KUKA KRL program: EPS_2_26115_SA6997_A_20260219035528.src

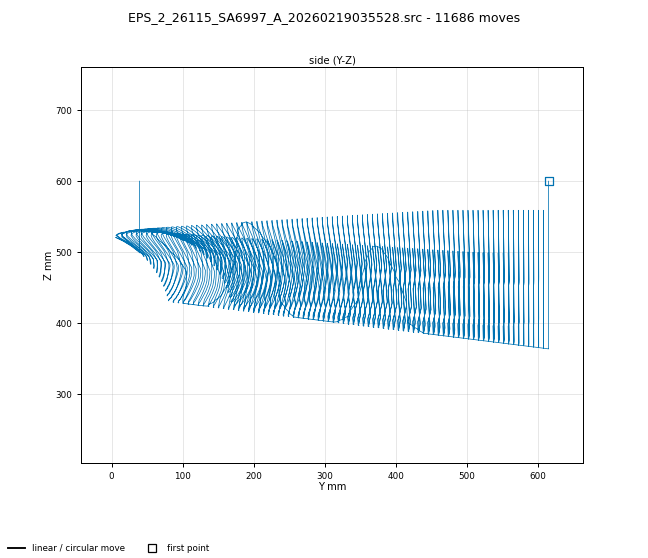
[picture p0: tool path of EPS_2_26115_SA6997_A_20260219035528.src, 11686 of 11688 moves have a stored position in this frame; points joined in program order, loops and branches not executed]
&ACCESS RVP
&REL 4
&COMMENT QRS 19112012
&PARAM EDITMASK = *
DEF PART()
EXT BAS (BAS_COMMAND :IN,REAL :IN )
INT I
BAS (#INITMOV,0 )

;KUKA QRS Post kuka4.cps  Date:22-06-2017 !

File_ID=3052

QRS_PRE_INIT()

;Init var - Until changes are made in qrs_pre_init
Outlet_Square_prg=0
Inlet_1_Square_prg=0
Inlet_2_Square_prg=0
Inlet_3_Square_prg=0
Inlet_4_Square_prg=0
Inlet_5_Square_prg=0

Outlet_1={X 0.000, Y 460.000, Z 458.500, B 0.000, E1 0.000 }
Inlet_1={X 0.000, Y 525.210, Z 398.500, B 0.000, E1 212.000 }
Outlet_1_type=201
Inlet_1_type=201
;QRS#1=Sidecore dimensions
;QRS#2=200-8" PVC SDR 35 Cut Back
;QRS#3=200-8" PVC SDR 35
;QRS#4=
;QRS#5=
;QRS#6=
;QRS#7=
;QRS#8=
;QRS#9=12-08 PSX
;QRS#10=12-08 PSX
;QRS#11=
;QRS#12=
;QRS#13=
;QRS#14=
;QRS#15=
;QRS#16=1220x127x838 2,75'
;QRS#17=EPS Height
;QRS#18=559
;QRS#19=*
;QRS#20= UPDATED VERSION 22-06-2017
;QRS#21=*
Outlet_Square=0100
Inlet_1_Square=0100
Inlet_2_Square=0
Inlet_3_Square=0
Inlet_4_Square=0
Inlet_5_Square=0
Mill_Square=1
Outlet_Square_Prg=214
Inlet_1_Square_prg=204

QRS_INIT()

$ADVANCE=5

; T1
PTP {E1 173.601,E2 173.601}
PTP {X 0,Y 615.495,A -85,B 0,C 180,E1 173.601,E2 173.601,E3 0,E4 0,E5 0,E6 0}
QRS_SPEED_INIT()
LIN {X 0,Y 615.495,Z 600,A -85,B 0,C 180,E1 173.601,E2 173.601,E3 0,E4 0,E5 0,E6 0} C_VEL
LIN {X 0,Y 615.495,Z 373.874,A -85,B 0,C 180,E1 173.601,E2 173.601} C_VEL
LIN {X 0,Y 615.495,Z 365.698,A -85,B 0,C 180,E1 173.601,E2 173.601} C_VEL
LIN {X 0,Y 615.482,Z 363.698,A -85,B 0,C 180,E1 173.415,E2 173.415} C_VEL
LIN {X 0,Y 615.496,Z 363.698,A -85,B 0,C 180,E1 170.801,E2 170.801} C_VEL
LIN {X 0,Y 615.477,Z 363.7,A -85,B 0,C 180,E1 168.139,E2 168.139} C_VEL
LIN {X 0,Y 615.479,Z 363.699,A -85,B 0,C 180,E1 165.451,E2 165.451} C_VEL
LIN {X 0,Y 615.484,Z 363.7,A -85,B 0,C 180,E1 162.729,E2 162.729} C_VEL
LIN {X 0,Y 615.472,Z 363.701,A -85,B 0,C 180,E1 159.967,E2 159.967} C_VEL
LIN {X 0,Y 615.492,Z 363.698,A -85,B 0,C 180,E1 157.155,E2 157.155} C_VEL
LIN {X 0,Y 615.482,Z 363.7,A -85,B 0,C 180,E1 154.284,E2 154.284} C_VEL
LIN {X 0,Y 615.49,Z 363.697,A -85,B 0,C 180,E1 151.547,E2 151.547} C_VEL
LIN {X 0,Y 615.485,Z 363.698,A -85,B 0,C 180,E1 148.912,E2 148.912} C_VEL
LIN {X 0,Y 615.484,Z 363.701,A -85,B 0,C 180,E1 146.464,E2 146.464} C_VEL
LIN {X 0,Y 615.492,Z 363.7,A -85,B 0,C 180,E1 144.164,E2 144.164} C_VEL
LIN {X 0,Y 615.491,Z 363.701,A -85,B 0,C 180,E1 141.931,E2 141.931} C_VEL
LIN {X 0,Y 615.48,Z 363.699,A -85,B 0,C 180,E1 138.905,E2 138.905} C_VEL
LIN {X 0,Y 615.482,Z 363.698,A -85,B 0,C 180,E1 136.002,E2 136.002} C_VEL
LIN {X 0,Y 615.489,Z 363.702,A -85,B 0,C 180,E1 133.047,E2 133.047} C_VEL
LIN {X 0,Y 615.479,Z 363.701,A -85,B 0,C 180,E1 130.606,E2 130.606} C_VEL
LIN {X 0,Y 615.475,Z 363.699,A -85,B 0,C 180,E1 128.01,E2 128.01} C_VEL
LIN {X 0,Y 615.498,Z 363.695,A -85,B 0,C 180,E1 125.614,E2 125.614} C_VEL
LIN {X 0,Y 615.487,Z 363.7,A -85,B 0,C 180,E1 123.235,E2 123.235} C_VEL
LIN {X 0,Y 615.495,Z 363.7,A -85,B 0,C 180,E1 120.918,E2 120.918} C_VEL
LIN {X 0,Y 615.485,Z 363.7,A -85,B 0,C 180,E1 118.449,E2 118.449} C_VEL
LIN {X 0,Y 615.496,Z 363.696,A -85,B 0,C 180,E1 115.57,E2 115.57} C_VEL
LIN {X 0,Y 615.479,Z 363.7,A -85,B 0,C 180,E1 112.844,E2 112.844} C_VEL
LIN {X 0,Y 615.481,Z 363.7,A -85,B 0,C 180,E1 110.032,E2 110.032} C_VEL
LIN {X 0,Y 615.475,Z 363.701,A -85,B 0,C 180,E1 107.27,E2 107.27} C_VEL
LIN {X 0,Y 615.478,Z 363.7,A -85,B 0,C 180,E1 104.549,E2 104.549} C_VEL
LIN {X 0,Y 615.492,Z 363.698,A -85,B 0,C 180,E1 101.86,E2 101.86} C_VEL
LIN {X 0,Y 615.472,Z 363.7,A -85,B 0,C 180,E1 99.199,E2 99.199} C_VEL
LIN {X 0,Y 615.493,Z 363.701,A -85,B 0,C 180,E1 96.556,E2 96.556} C_VEL
LIN {X 0,Y 615.492,Z 363.696,A -85,B 0,C 180,E1 93.928,E2 93.928} C_VEL
LIN {X 0,Y 615.491,Z 363.758,A -85,B 0,C 180,E1 93.273,E2 93.273} C_VEL
LIN {X 0,Y 615.489,Z 366.912,A -85,B 0,C 180,E1 90.654,E2 90.654} C_VEL
LIN {X 0,Y 615.499,Z 370.079,A -85,B 0,C 180,E1 88.037,E2 88.037} C_VEL
LIN {X 0,Y 615.458,Z 373.445,A -85,B 0,C 180,E1 85.415,E2 85.415} C_VEL
LIN {X 0,Y 615.488,Z 376.887,A -85,B 0,C 180,E1 82.784,E2 82.784} C_VEL
LIN {X 0,Y 615.495,Z 380.418,A -85,B 0,C 180,E1 80.138,E2 80.138} C_VEL
LIN {X 0,Y 615.475,Z 384.071,A -85,B 0,C 180,E1 77.47,E2 77.47} C_VEL
LIN {X 0,Y 615.479,Z 387.794,A -85,B 0,C 180,E1 74.774,E2 74.774} C_VEL
LIN {X 0,Y 615.49,Z 391.632,A -85,B 0,C 180,E1 72.043,E2 72.043} C_VEL
LIN {X 0,Y 615.492,Z 395.191,A -85,B 0,C 180,E1 69.542,E2 69.542} C_VEL
LIN {X 0,Y 615.481,Z 409.079,A -85,B 0,C 180,E1 69.226,E2 69.226} C_VEL
LIN {X 0,Y 615.467,Z 420.927,A -85,B 0,C 180,E1 68.831,E2 68.831} C_VEL
LIN {X 0,Y 615.492,Z 432.681,A -85,B 0,C 180,E1 68.305,E2 68.305} C_VEL
LIN {X 0,Y 615.492,Z 443.951,A -85,B 0,C 180,E1 67.654,E2 67.654} C_VEL
LIN {X 0,Y 615.499,Z 454.538,A -85,B 0,C 180,E1 66.89,E2 66.89} C_VEL
LIN {X 0,Y 615.497,Z 463.408,A -85,B 0,C 180,E1 66.104,E2 66.104} C_VEL
LIN {X 0,Y 615.496,Z 471.812,A -85,B 0,C 180,E1 65.189,E2 65.189} C_VEL
LIN {X 0,Y 615.497,Z 479.85,A -85,B 0,C 180,E1 64.103,E2 64.103} C_VEL
LIN {X 0,Y 615.498,Z 484.877,A -85,B 0,C 180,E1 63.256,E2 63.256} C_VEL
LIN {X 0,Y 615.495,Z 490.382,A -85,B 0,C 180,E1 62.086,E2 62.086} C_VEL
LIN {X 0,Y 615.497,Z 494.172,A -85,B 0,C 180,E1 60.969,E2 60.969} C_VEL
LIN {X 0,Y 615.494,Z 496.737,A -85,B 0,C 180,E1 59.841,E2 59.841} C_VEL
LIN {X 0,Y 615.496,Z 497.959,A -85,B 0,C 180,E1 58.913,E2 58.913} C_VEL
LIN {X 0,Y 615.494,Z 498.327,A -85,B 0,C 180,E1 57.669,E2 57.669} C_VEL
LIN {X 0,Y 615.496,Z 497.367,A -85,B 0,C 180,E1 56.465,E2 56.465} C_VEL
LIN {X 0,Y 615.491,Z 494.83,A -85,B 0,C 180,E1 55.186,E2 55.186} C_VEL
LIN {X 0,Y 615.493,Z 491.663,A -85,B 0,C 180,E1 54.166,E2 54.166} C_VEL
LIN {X 0,Y 615.495,Z 486.974,A -85,B 0,C 180,E1 53.063,E2 53.063} C_VEL
LIN {X 0,Y 615.495,Z 480.669,A -85,B 0,C 180,E1 51.933,E2 51.933} C_VEL
LIN {X 0,Y 615.498,Z 473.586,A -85,B 0,C 180,E1 50.937,E2 50.937} C_VEL
LIN {X 0,Y 615.498,Z 464.435,A -85,B 0,C 180,E1 49.91,E2 49.91} C_VEL
LIN {X 0,Y 615.499,Z 454.637,A -85,B 0,C 180,E1 49.028,E2 49.028} C_VEL
LIN {X 0,Y 615.473,Z 443.526,A -85,B 0,C 180,E1 48.228,E2 48.228} C_VEL
LIN {X 0,Y 615.419,Z 433.407,A -85,B 0,C 180,E1 47.642,E2 47.642} C_VEL
LIN {X 0,Y 615.427,Z 421.147,A -85,B 0,C 180,E1 47.086,E2 47.086} C_VEL
LIN {X 0,Y 615.473,Z 408.287,A -85,B 0,C 180,E1 46.662,E2 46.662} C_VEL
LIN {X 0,Y 615.474,Z 395.186,A -85,B 0,C 180,E1 46.361,E2 46.361} C_VEL
LIN {X 0,Y 615.437,Z 391.826,A -85,B 0,C 180,E1 43.994,E2 43.994} C_VEL
LIN {X 0,Y 615.43,Z 388.283,A -85,B 0,C 180,E1 41.479,E2 41.479} C_VEL
LIN {X 0,Y 615.485,Z 384.702,A -85,B 0,C 180,E1 38.905,E2 38.905} C_VEL
LIN {X 0,Y 615.474,Z 381.317,A -85,B 0,C 180,E1 36.426,E2 36.426} C_VEL
LIN {X 0,Y 615.45,Z 378.084,A -85,B 0,C 180,E1 34.025,E2 34.025} C_VEL
LIN {X 0,Y 615.457,Z 374.994,A -85,B 0,C 180,E1 31.687,E2 31.687} C_VEL
LIN {X 0,Y 615.481,Z 372.039,A -85,B 0,C 180,E1 29.407,E2 29.407} C_VEL
LIN {X 0,Y 615.493,Z 368.347,A -85,B 0,C 180,E1 26.444,E2 26.444} C_VEL
LIN {X 0,Y 615.491,Z 365.458,A -85,B 0,C 180,E1 24.011,E2 24.011} C_VEL
LIN {X 0,Y 615.471,Z 363.7,A -85,B 0,C 180,E1 22.345,E2 22.345} C_VEL
LIN {X 0,Y 615.479,Z 363.7,A -85,B 0,C 180,E1 20.033,E2 20.033} C_VEL
LIN {X 0,Y 615.476,Z 363.698,A -85,B 0,C 180,E1 17.271,E2 17.271} C_VEL
LIN {X 0,Y 615.488,Z 363.697,A -85,B 0,C 180,E1 14.549,E2 14.549} C_VEL
LIN {X 0,Y 615.485,Z 363.702,A -85,B 0,C 180,E1 11.861,E2 11.861} C_VEL
LIN {X 0,Y 615.495,Z 363.697,A -85,B 0,C 180,E1 9.199,E2 9.199} C_VEL
LIN {X 0,Y 615.471,Z 363.7,A -85,B 0,C 180,E1 6.557,E2 6.557} C_VEL
LIN {X 0,Y 615.466,Z 363.7,A -85,B 0,C 180,E1 3.929,E2 3.929} C_VEL
LIN {X 0,Y 615.477,Z 363.698,A -85,B 0,C 180,E1 1.309,E2 1.309} C_VEL
LIN {X 0,Y 615.493,Z 363.697,A -85,B 0,C 180,E1 -1.309,E2 -1.309} C_VEL
LIN {X 0,Y 615.487,Z 363.702,A -85,B 0,C 180,E1 -3.928,E2 -3.928} C_VEL
LIN {X 0,Y 615.494,Z 363.697,A -85,B 0,C 180,E1 -6.591,E2 -6.591} C_VEL
LIN {X 0,Y 615.477,Z 363.698,A -85,B 0,C 180,E1 -9.199,E2 -9.199} C_VEL
LIN {X 0,Y 615.466,Z 363.7,A -85,B 0,C 180,E1 -11.861,E2 -11.861} C_VEL
LIN {X 0,Y 615.476,Z 363.699,A -85,B 0,C 180,E1 -14.549,E2 -14.549} C_VEL
LIN {X 0,Y 615.499,Z 363.7,A -85,B 0,C 180,E1 -17.27,E2 -17.27} C_VEL
LIN {X 0,Y 615.477,Z 363.699,A -85,B 0,C 180,E1 -20.033,E2 -20.033} C_VEL
LIN {X 0,Y 615.495,Z 363.694,A -85,B 0,C 180,E1 -22.844,E2 -22.844} C_VEL
LIN {X 0,Y 615.495,Z 363.7,A -85,B 0,C 180,E1 -25.715,E2 -25.715} C_VEL
LIN {X 0,Y 615.491,Z 363.695,A -85,B 0,C 180,E1 -28.658,E2 -28.658} C_VEL
LIN {X 0,Y 615.485,Z 363.7,A -85,B 0,C 180,E1 -31.686,E2 -31.686} C_VEL
LIN {X 0,Y 615.479,Z 363.7,A -85,B 0,C 180,E1 -34.023,E2 -34.023} C_VEL
LIN {X 0,Y 615.479,Z 363.7,A -85,B 0,C 180,E1 -36.425,E2 -36.425} C_VEL
LIN {X 0,Y 615.496,Z 363.7,A -85,B 0,C 180,E1 -39.064,E2 -39.064} C_VEL
LIN {X 0,Y 615.492,Z 363.701,A -85,B 0,C 180,E1 -41.474,E2 -41.474} C_VEL
LIN {X 0,Y 615.493,Z 363.697,A -85,B 0,C 180,E1 -44.149,E2 -44.149} C_VEL
LIN {X 0,Y 615.473,Z 363.698,A -85,B 0,C 180,E1 -46.954,E2 -46.954} C_VEL
LIN {X 0,Y 615.466,Z 363.7,A -85,B 0,C 180,E1 -49.393,E2 -49.393} C_VEL
LIN {X 0,Y 615.469,Z 363.7,A -85,B 0,C 180,E1 -51.991,E2 -51.991} C_VEL
LIN {X 0,Y 615.494,Z 363.819,A -85,B 0,C 180,E1 -54.536,E2 -54.536} C_VEL
LIN {X 0,Y 615.444,Z 372.581,A -85,B 0,C 180,E1 -57.152,E2 -57.152} C_VEL
LIN {X 0,Y 615.423,Z 380.515,A -85,B 0,C 180,E1 -59.458,E2 -59.458} C_VEL
LIN {X 0,Y 615.479,Z 389.757,A -85,B 0,C 180,E1 -62.085,E2 -62.085} C_VEL
LIN {X 0,Y 615.455,Z 399.273,A -85,B 0,C 180,E1 -64.72,E2 -64.72} C_VEL
LIN {X 0,Y 615.46,Z 408.239,A -85,B 0,C 180,E1 -67.155,E2 -67.155} C_VEL
LIN {X 0,Y 615.489,Z 416.801,A -85,B 0,C 180,E1 -69.443,E2 -69.443} C_VEL
LIN {X 0,Y 615.487,Z 428.015,A -85,B 0,C 180,E1 -72.387,E2 -72.387} C_VEL
LIN {X 0,Y 615.482,Z 438.542,A -85,B 0,C 180,E1 -75.113,E2 -75.113} C_VEL
LIN {X 0,Y 615.469,Z 449.085,A -85,B 0,C 180,E1 -77.804,E2 -77.804} C_VEL
LIN {X 0,Y 615.495,Z 451.209,A -85,B 0,C 180,E1 -78.348,E2 -78.348} C_VEL
LIN {X 0,Y 615.497,Z 465.824,A -85,B 0,C 180,E1 -78.64,E2 -78.64} C_VEL
LIN {X 0,Y 615.457,Z 478.917,A -85,B 0,C 180,E1 -79.049,E2 -79.049} C_VEL
LIN {X 0,Y 615.451,Z 490.773,A -85,B 0,C 180,E1 -79.556,E2 -79.556} C_VEL
LIN {X 0,Y 615.496,Z 501.387,A -85,B 0,C 180,E1 -80.138,E2 -80.138} C_VEL
LIN {X 0,Y 615.498,Z 512.232,A -85,B 0,C 180,E1 -80.884,E2 -80.884} C_VEL
LIN {X 0,Y 615.497,Z 522.812,A -85,B 0,C 180,E1 -81.794,E2 -81.794} C_VEL
LIN {X 0,Y 615.498,Z 530.606,A -85,B 0,C 180,E1 -82.62,E2 -82.62} C_VEL
LIN {X 0,Y 615.496,Z 538.203,A -85,B 0,C 180,E1 -83.608,E2 -83.608} C_VEL
LIN {X 0,Y 615.498,Z 545.204,A -85,B 0,C 180,E1 -84.759,E2 -84.759} C_VEL
LIN {X 0,Y 615.494,Z 549.851,A -85,B 0,C 180,E1 -85.744,E2 -85.744} C_VEL
LIN {X 0,Y 615.494,Z 553.398,A -85,B 0,C 180,E1 -86.727,E2 -86.727} C_VEL
LIN {X 0,Y 615.497,Z 555.233,A -85,B 0,C 180,E1 -87.382,E2 -87.382} C_VEL
LIN {X 0,Y 615.499,Z 556.607,A -85,B 0,C 180,E1 -88.037,E2 -88.037} C_VEL
LIN {X 0,Y 615.496,Z 558.173,A -85,B 0,C 180,E1 -89.346,E2 -89.346} C_VEL
LIN {X 0,Y 615.494,Z 558.389,A -85,B 0,C 180,E1 -90,E2 -90} C_VEL
LIN {X 0,Y 615.495,Z 557.58,A -85,B 0,C 180,E1 -91.308,E2 -91.308} C_VEL
LIN {X 0,Y 615.499,Z 556.608,A -85,B 0,C 180,E1 -91.963,E2 -91.963} C_VEL
LIN {X 0,Y 615.497,Z 555.233,A -85,B 0,C 180,E1 -92.618,E2 -92.618} C_VEL
LIN {X 0,Y 615.496,Z 552.35,A -85,B 0,C 180,E1 -93.6,E2 -93.6} C_VEL
LIN {X 0,Y 615.498,Z 548.443,A -85,B 0,C 180,E1 -94.584,E2 -94.584} C_VEL
LIN {X 0,Y 615.499,Z 543.406,A -85,B 0,C 180,E1 -95.569,E2 -95.569} C_VEL
LIN {X 0,Y 615.497,Z 536.87,A -85,B 0,C 180,E1 -96.583,E2 -96.583} C_VEL
LIN {X 0,Y 615.497,Z 529.136,A -85,B 0,C 180,E1 -97.545,E2 -97.545} C_VEL
LIN {X 0,Y 615.498,Z 521.048,A -85,B 0,C 180,E1 -98.371,E2 -98.371} C_VEL
LIN {X 0,Y 615.499,Z 511.172,A -85,B 0,C 180,E1 -99.198,E2 -99.198} C_VEL
LIN {X 0,Y 615.487,Z 499.988,A -85,B 0,C 180,E1 -99.945,E2 -99.945} C_VEL
LIN {X 0,Y 615.449,Z 489.037,A -85,B 0,C 180,E1 -100.527,E2 -100.527} C_VEL
LIN {X 0,Y 615.463,Z 476.744,A -85,B 0,C 180,E1 -101.032,E2 -101.032} C_VEL
LIN {X 0,Y 615.498,Z 464.08,A -85,B 0,C 180,E1 -101.401,E2 -101.401} C_VEL
LIN {X 0,Y 615.494,Z 451.21,A -85,B 0,C 180,E1 -101.651,E2 -101.651} C_VEL
LIN {X 0,Y 615.471,Z 441.068,A -85,B 0,C 180,E1 -104.241,E2 -104.241} C_VEL
LIN {X 0,Y 615.49,Z 430.642,A -85,B 0,C 180,E1 -106.928,E2 -106.928} C_VEL
LIN {X 0,Y 615.484,Z 420.106,A -85,B 0,C 180,E1 -109.684,E2 -109.684} C_VEL
LIN {X 0,Y 615.491,Z 410.086,A -85,B 0,C 180,E1 -112.346,E2 -112.346} C_VEL
LIN {X 0,Y 615.445,Z 400.327,A -85,B 0,C 180,E1 -114.993,E2 -114.993} C_VEL
LIN {X 0,Y 615.476,Z 391.078,A -85,B 0,C 180,E1 -117.545,E2 -117.545} C_VEL
LIN {X 0,Y 615.439,Z 381.837,A -85,B 0,C 180,E1 -120.162,E2 -120.162} C_VEL
LIN {X 0,Y 615.433,Z 373.906,A -85,B 0,C 180,E1 -122.46,E2 -122.46} C_VEL
LIN {X 0,Y 615.461,Z 365.97,A -85,B 0,C 180,E1 -124.816,E2 -124.816} C_VEL
LIN {X 0,Y 615.495,Z 363.696,A -85,B 0,C 180,E1 -125.514,E2 -125.514} C_VEL
LIN {X 0,Y 615.482,Z 363.698,A -85,B 0,C 180,E1 -128.068,E2 -128.068} C_VEL
LIN {X 0,Y 615.483,Z 363.702,A -85,B 0,C 180,E1 -130.606,E2 -130.606} C_VEL
LIN {X 0,Y 615.491,Z 363.697,A -85,B 0,C 180,E1 -133.243,E2 -133.243} C_VEL
LIN {X 0,Y 615.487,Z 363.699,A -85,B 0,C 180,E1 -136.001,E2 -136.001} C_VEL
LIN {X 0,Y 615.49,Z 363.701,A -85,B 0,C 180,E1 -138.526,E2 -138.526} C_VEL
LIN {X 0,Y 615.486,Z 363.697,A -85,B 0,C 180,E1 -141.095,E2 -141.095} C_VEL
LIN {X 0,Y 615.49,Z 363.696,A -85,B 0,C 180,E1 -143.575,E2 -143.575} C_VEL
LIN {X 0,Y 615.486,Z 363.699,A -85,B 0,C 180,E1 -145.978,E2 -145.978} C_VEL
LIN {X 0,Y 615.486,Z 363.701,A -85,B 0,C 180,E1 -148.314,E2 -148.314} C_VEL
LIN {X 0,Y 615.49,Z 363.702,A -85,B 0,C 180,E1 -150.594,E2 -150.594} C_VEL
LIN {X 0,Y 615.489,Z 363.697,A -85,B 0,C 180,E1 -153.556,E2 -153.556} C_VEL
LIN {X 0,Y 615.483,Z 363.701,A -85,B 0,C 180,E1 -155.99,E2 -155.99} C_VEL
LIN {X 0,Y 615.487,Z 363.699,A -85,B 0,C 180,E1 -158.568,E2 -158.568} C_VEL
LIN {X 0,Y 615.494,Z 363.697,A -85,B 0,C 180,E1 -161.39,E2 -161.39} C_VEL
LIN {X 0,Y 615.483,Z 363.7,A -85,B 0,C 180,E1 -164.095,E2 -164.095} C_VEL
LIN {X 0,Y 615.478,Z 363.699,A -85,B 0,C 180,E1 -166.799,E2 -166.799} C_VEL
LIN {X 0,Y 615.49,Z 363.701,A -85,B 0,C 180,E1 -169.473,E2 -169.473} C_VEL
LIN {X 0,Y 615.472,Z 363.7,A -85,B 0,C 180,E1 -172.124,E2 -172.124} C_VEL
LIN {X 0,Y 615.479,Z 363.701,A -85,B 0,C 180,E1 -174.759,E2 -174.759} C_VEL
LIN {X 0,Y 615.479,Z 363.701,A -85,B 0,C 180,E1 -177.382,E2 -177.382} C_VEL
LIN {X 0,Y 615.472,Z 363.7,A -85,B 0,C 180,E1 -180,E2 -180} C_VEL
LIN {X 0,Y 615.488,Z 363.701,A -85,B 0,C 180,E1 -182.618,E2 -182.618} C_VEL
LIN {X 0,Y 615.479,Z 363.7,A -85,B 0,C 180,E1 -185.241,E2 -185.241} C_VEL
LIN {X 0,Y 615.482,Z 363.698,A -85,B 0,C 180,E1 -186.585,E2 -186.585} C_VEL
LIN {X 0,Y 614.813,Z 363.845,A -85,B 0,C 180,E1 -187.131,E2 -187.131} C_VEL
LIN {X 0,Y 611.986,Z 364.256,A -85,B 0,C 180,E1 -188.017,E2 -188.017} C_VEL
LIN {X 0,Y 609.594,Z 364.568,A -85,B 0,C 180,E1 -188.73,E2 -188.73} C_VEL
LIN {X 0,Y 608.553,Z 364.686,A -85,B 0,C 180,E1 -189.279,E2 -189.279} C_VEL
LIN {X 0,Y 608.46,Z 364.695,A -85,B 0,C 180,E1 -189.466,E2 -189.466} C_VEL
LIN {X 0,Y 608.455,Z 364.695,A -85,B 0,C 180,E1 -192,E2 -192} C_VEL
LIN {X 0,Y 608.467,Z 364.695,A -85,B 0,C 180,E1 -194.721,E2 -194.721} C_VEL
LIN {X 0,Y 608.447,Z 364.696,A -85,B 0,C 180,E1 -197.477,E2 -197.477} C_VEL
LIN {X 0,Y 608.459,Z 364.696,A -85,B 0,C 180,E1 -200.274,E2 -200.274} C_VEL
LIN {X 0,Y 608.453,Z 364.695,A -85,B 0,C 180,E1 -203.124,E2 -203.124} C_VEL
LIN {X 0,Y 608.464,Z 364.695,A -85,B 0,C 180,E1 -205.722,E2 -205.722} C_VEL
LIN {X 0,Y 608.452,Z 364.697,A -85,B 0,C 180,E1 -208.267,E2 -208.267} C_VEL
LIN {X 0,Y 608.467,Z 364.695,A -85,B 0,C 180,E1 -210.545,E2 -210.545} C_VEL
LIN {X 0,Y 608.449,Z 364.696,A -85,B 0,C 180,E1 -212.88,E2 -212.88} C_VEL
LIN {X 0,Y 608.442,Z 364.696,A -85,B 0,C 180,E1 -215.278,E2 -215.278} C_VEL
LIN {X 0,Y 608.467,Z 364.693,A -85,B 0,C 180,E1 -217.747,E2 -217.747} C_VEL
LIN {X 0,Y 608.451,Z 364.699,A -85,B 0,C 180,E1 -220.33,E2 -220.33} C_VEL
LIN {X 0,Y 608.46,Z 364.694,A -85,B 0,C 180,E1 -223.309,E2 -223.309} C_VEL
LIN {X 0,Y 608.477,Z 364.693,A -85,B 0,C 180,E1 -226.133,E2 -226.133} C_VEL
LIN {X 0,Y 608.459,Z 364.695,A -85,B 0,C 180,E1 -228.825,E2 -228.825} C_VEL
LIN {X 0,Y 608.462,Z 364.697,A -85,B 0,C 180,E1 -231.413,E2 -231.413} C_VEL
LIN {X 0,Y 608.477,Z 364.692,A -85,B 0,C 180,E1 -233.951,E2 -233.951} C_VEL
LIN {X 0,Y 608.472,Z 364.693,A -85,B 0,C 180,E1 -236.331,E2 -236.331} C_VEL
LIN {X 0,Y 608.479,Z 364.692,A -85,B 0,C 180,E1 -238.728,E2 -238.728} C_VEL
LIN {X 0,Y 608.473,Z 364.696,A -85,B 0,C 180,E1 -241.381,E2 -241.381} C_VEL
LIN {X 0,Y 608.482,Z 364.692,A -85,B 0,C 180,E1 -244.278,E2 -244.278} C_VEL
LIN {X 0,Y 608.449,Z 364.699,A -85,B 0,C 180,E1 -246.877,E2 -246.877} C_VEL
LIN {X 0,Y 608.461,Z 364.695,A -85,B 0,C 180,E1 -249.324,E2 -249.324} C_VEL
LIN {X 0,Y 608.452,Z 364.695,A -85,B 0,C 180,E1 -251.829,E2 -251.829} C_VEL
LIN {X 0,Y 608.47,Z 364.696,A -85,B 0,C 180,E1 -254.595,E2 -254.595} C_VEL
LIN {X 0,Y 608.465,Z 364.693,A -85,B 0,C 180,E1 -257.323,E2 -257.323} C_VEL
LIN {X 0,Y 608.464,Z 364.695,A -85,B 0,C 180,E1 -260.023,E2 -260.023} C_VEL
LIN {X 0,Y 608.443,Z 364.697,A -85,B 0,C 180,E1 -262.701,E2 -262.701} C_VEL
LIN {X 0,Y 608.447,Z 364.696,A -85,B 0,C 180,E1 -265.363,E2 -265.363} C_VEL
LIN {X 0,Y 608.453,Z 364.697,A -85,B 0,C 180,E1 -266.689,E2 -266.689} C_VEL
LIN {X 0,Y 608.438,Z 367.735,A -85,B 0,C 180,E1 -269.338,E2 -269.338} C_VEL
LIN {X 0,Y 608.465,Z 370.901,A -85,B 0,C 180,E1 -271.986,E2 -271.986} C_VEL
LIN {X 0,Y 608.411,Z 374.282,A -85,B 0,C 180,E1 -274.638,E2 -274.638} C_VEL
LIN {X 0,Y 608.433,Z 377.752,A -85,B 0,C 180,E1 -277.3,E2 -277.3} C_VEL
LIN {X 0,Y 608.427,Z 381.321,A -85,B 0,C 180,E1 -279.978,E2 -279.978} C_VEL
LIN {X 0,Y 608.406,Z 384.989,A -85,B 0,C 180,E1 -282.678,E2 -282.678} C_VEL
LIN {X 0,Y 608.407,Z 387.806,A -85,B 0,C 180,E1 -284.722,E2 -284.722} C_VEL
LIN {X 0,Y 608.405,Z 391.653,A -85,B 0,C 180,E1 -287.478,E2 -287.478} C_VEL
LIN {X 0,Y 608.419,Z 395.679,A -85,B 0,C 180,E1 -290.325,E2 -290.325} C_VEL
LIN {X 0,Y 608.54,Z 410.666,A -85,B 0,C 180,E1 -290.685,E2 -290.685} C_VEL
LIN {X 0,Y 608.491,Z 422.804,A -85,B 0,C 180,E1 -291.113,E2 -291.113} C_VEL
LIN {X 0,Y 608.52,Z 434.966,A -85,B 0,C 180,E1 -291.689,E2 -291.689} C_VEL
LIN {X 0,Y 608.499,Z 446.745,A -85,B 0,C 180,E1 -292.404,E2 -292.404} C_VEL
LIN {X 0,Y 608.467,Z 457.265,A -85,B 0,C 180,E1 -293.213,E2 -293.213} C_VEL
LIN {X 0,Y 608.464,Z 467.103,A -85,B 0,C 180,E1 -294.149,E2 -294.149} C_VEL
LIN {X 0,Y 608.458,Z 475.284,A -85,B 0,C 180,E1 -295.117,E2 -295.117} C_VEL
LIN {X 0,Y 608.449,Z 482.724,A -85,B 0,C 180,E1 -296.219,E2 -296.219} C_VEL
LIN {X 0,Y 608.437,Z 487.966,A -85,B 0,C 180,E1 -297.199,E2 -297.199} C_VEL
LIN {X 0,Y 608.441,Z 492.405,A -85,B 0,C 180,E1 -298.267,E2 -298.267} C_VEL
LIN {X 0,Y 608.427,Z 494.809,A -85,B 0,C 180,E1 -299.022,E2 -299.022} C_VEL
LIN {X 0,Y 608.44,Z 497.044,A -85,B 0,C 180,E1 -299.966,E2 -299.966} C_VEL
LIN {X 0,Y 608.424,Z 498.699,A -85,B 0,C 180,E1 -301.263,E2 -301.263} C_VEL
LIN {X 0,Y 608.419,Z 498.896,A -85,B 0,C 180,E1 -302.515,E2 -302.515} C_VEL
LIN {X 0,Y 608.421,Z 497.706,A -85,B 0,C 180,E1 -303.727,E2 -303.727} C_VEL
LIN {X 0,Y 608.419,Z 495.256,A -85,B 0,C 180,E1 -304.901,E2 -304.901} C_VEL
LIN {X 0,Y 608.427,Z 491.401,A -85,B 0,C 180,E1 -306.093,E2 -306.093} C_VEL
LIN {X 0,Y 608.435,Z 486.692,A -85,B 0,C 180,E1 -307.153,E2 -307.153} C_VEL
LIN {X 0,Y 608.456,Z 480.454,A -85,B 0,C 180,E1 -308.238,E2 -308.238} C_VEL
LIN {X 0,Y 608.445,Z 472.743,A -85,B 0,C 180,E1 -309.294,E2 -309.294} C_VEL
LIN {X 0,Y 608.477,Z 464.659,A -85,B 0,C 180,E1 -310.192,E2 -310.192} C_VEL
LIN {X 0,Y 608.487,Z 455.047,A -85,B 0,C 180,E1 -311.063,E2 -311.063} C_VEL
LIN {X 0,Y 608.472,Z 444.03,A -85,B 0,C 180,E1 -311.865,E2 -311.865} C_VEL
LIN {X 0,Y 608.423,Z 433.268,A -85,B 0,C 180,E1 -312.494,E2 -312.494} C_VEL
LIN {X 0,Y 608.453,Z 421.105,A -85,B 0,C 180,E1 -313.046,E2 -313.046} C_VEL
LIN {X 0,Y 608.515,Z 408.391,A -85,B 0,C 180,E1 -313.469,E2 -313.469} C_VEL
LIN {X 0,Y 608.394,Z 395.673,A -85,B 0,C 180,E1 -313.769,E2 -313.769} C_VEL
LIN {X 0,Y 608.375,Z 391.531,A -85,B 0,C 180,E1 -316.7,E2 -316.7} C_VEL
LIN {X 0,Y 608.386,Z 388.571,A -85,B 0,C 180,E1 -318.817,E2 -318.817} C_VEL
LIN {X 0,Y 608.382,Z 384.502,A -85,B 0,C 180,E1 -321.769,E2 -321.769} C_VEL
LIN {X 0,Y 608.399,Z 381.528,A -85,B 0,C 180,E1 -323.959,E2 -323.959} C_VEL
LIN {X 0,Y 608.404,Z 378.368,A -85,B 0,C 180,E1 -326.325,E2 -326.325} C_VEL
LIN {X 0,Y 608.445,Z 375.212,A -85,B 0,C 180,E1 -328.731,E2 -328.731} C_VEL
LIN {X 0,Y 608.418,Z 371.374,A -85,B 0,C 180,E1 -331.731,E2 -331.731} C_VEL
LIN {X 0,Y 608.454,Z 368.32,A -85,B 0,C 180,E1 -334.281,E2 -334.281} C_VEL
LIN {X 0,Y 608.449,Z 365.237,A -85,B 0,C 180,E1 -336.876,E2 -336.876} C_VEL
LIN {X 0,Y 608.452,Z 364.696,A -85,B 0,C 180,E1 -337.594,E2 -337.594} C_VEL
LIN {X 0,Y 608.462,Z 364.697,A -85,B 0,C 180,E1 -339.726,E2 -339.726} C_VEL
LIN {X 0,Y 608.447,Z 364.696,A -85,B 0,C 180,E1 -342.523,E2 -342.523} C_VEL
LIN {X 0,Y 608.476,Z 364.691,A -85,B 0,C 180,E1 -345.279,E2 -345.279} C_VEL
LIN {X 0,Y 608.458,Z 364.695,A -85,B 0,C 180,E1 -348,E2 -348} C_VEL
LIN {X 0,Y 608.473,Z 364.695,A -85,B 0,C 180,E1 -350.694,E2 -350.694} C_VEL
LIN {X 0,Y 608.449,Z 364.696,A -85,B 0,C 180,E1 -353.384,E2 -353.384} C_VEL
LIN {X 0,Y 608.437,Z 364.696,A -85,B 0,C 180,E1 -356.026,E2 -356.026} C_VEL
LIN {X 0,Y 608.461,Z 364.693,A -85,B 0,C 180,E1 -358.676,E2 -358.676} C_VEL
LIN {X 0,Y 608.475,Z 364.693,A -85,B 0,C 180,E1 -361.324,E2 -361.324} C_VEL
LIN {X 0,Y 608.454,Z 364.698,A -85,B 0,C 180,E1 -363.974,E2 -363.974} C_VEL
LIN {X 0,Y 608.47,Z 364.694,A -85,B 0,C 180,E1 -366.633,E2 -366.633} C_VEL
LIN {X 0,Y 608.462,Z 364.693,A -85,B 0,C 180,E1 -369.306,E2 -369.306} C_VEL
LIN {X 0,Y 608.448,Z 364.695,A -85,B 0,C 180,E1 -372,E2 -372} C_VEL
LIN {X 0,Y 608.464,Z 364.695,A -85,B 0,C 180,E1 -374.721,E2 -374.721} C_VEL
LIN {X 0,Y 608.454,Z 364.696,A -85,B 0,C 180,E1 -377.477,E2 -377.477} C_VEL
LIN {X 0,Y 608.456,Z 364.694,A -85,B 0,C 180,E1 -380.274,E2 -380.274} C_VEL
LIN {X 0,Y 608.452,Z 364.696,A -85,B 0,C 180,E1 -383.124,E2 -383.124} C_VEL
LIN {X 0,Y 608.449,Z 364.696,A -85,B 0,C 180,E1 -386.035,E2 -386.035} C_VEL
LIN {X 0,Y 608.476,Z 364.692,A -85,B 0,C 180,E1 -388.622,E2 -388.622} C_VEL
LIN {X 0,Y 608.439,Z 364.696,A -85,B 0,C 180,E1 -391.318,E2 -391.318} C_VEL
LIN {X 0,Y 608.439,Z 364.696,A -85,B 0,C 180,E1 -393.732,E2 -393.732} C_VEL
LIN {X 0,Y 608.44,Z 364.696,A -85,B 0,C 180,E1 -396.093,E2 -396.093} C_VEL
LIN {X 0,Y 608.472,Z 364.692,A -85,B 0,C 180,E1 -398.588,E2 -398.588} C_VEL
LIN {X 0,Y 608.462,Z 364.695,A -85,B 0,C 180,E1 -401.343,E2 -401.343} C_VEL
LIN {X 0,Y 608.461,Z 364.694,A -85,B 0,C 180,E1 -404.265,E2 -404.265} C_VEL
LIN {X 0,Y 608.442,Z 364.696,A -85,B 0,C 180,E1 -407.04,E2 -407.04} C_VEL
LIN {X 0,Y 608.45,Z 364.696,A -85,B 0,C 180,E1 -409.697,E2 -409.697} C_VEL
LIN {X 0,Y 608.455,Z 364.696,A -85,B 0,C 180,E1 -412.253,E2 -412.253} C_VEL
LIN {X 0,Y 608.492,Z 364.817,A -85,B 0,C 180,E1 -414.371,E2 -414.371} C_VEL
LIN {X 0,Y 608.495,Z 373.918,A -85,B 0,C 180,E1 -417.123,E2 -417.123} C_VEL
LIN {X 0,Y 608.454,Z 381.862,A -85,B 0,C 180,E1 -419.455,E2 -419.455} C_VEL
LIN {X 0,Y 608.492,Z 391.129,A -85,B 0,C 180,E1 -422.111,E2 -422.111} C_VEL
LIN {X 0,Y 608.446,Z 400.396,A -85,B 0,C 180,E1 -424.699,E2 -424.699} C_VEL
LIN {X 0,Y 608.443,Z 409.664,A -85,B 0,C 180,E1 -427.236,E2 -427.236} C_VEL
LIN {X 0,Y 608.465,Z 418.93,A -85,B 0,C 180,E1 -429.726,E2 -429.726} C_VEL
LIN {X 0,Y 608.458,Z 429.521,A -85,B 0,C 180,E1 -432.524,E2 -432.524} C_VEL
LIN {X 0,Y 608.439,Z 440.112,A -85,B 0,C 180,E1 -435.279,E2 -435.279} C_VEL
LIN {X 0,Y 608.425,Z 450.703,A -85,B 0,C 180,E1 -438,E2 -438} C_VEL
LIN {X 0,Y 608.441,Z 451.572,A -85,B 0,C 180,E1 -438.222,E2 -438.222} C_VEL
LIN {X 0,Y 608.548,Z 465.098,A -85,B 0,C 180,E1 -438.488,E2 -438.488} C_VEL
LIN {X 0,Y 608.489,Z 477.488,A -85,B 0,C 180,E1 -438.864,E2 -438.864} C_VEL
LIN {X 0,Y 608.473,Z 489.173,A -85,B 0,C 180,E1 -439.35,E2 -439.35} C_VEL
LIN {X 0,Y 608.486,Z 501.579,A -85,B 0,C 180,E1 -440.023,E2 -440.023} C_VEL
LIN {X 0,Y 608.483,Z 512.474,A -85,B 0,C 180,E1 -440.778,E2 -440.778} C_VEL
LIN {X 0,Y 608.475,Z 523.112,A -85,B 0,C 180,E1 -441.699,E2 -441.699} C_VEL
LIN {X 0,Y 608.471,Z 530.96,A -85,B 0,C 180,E1 -442.534,E2 -442.534} C_VEL
LIN {X 0,Y 608.461,Z 538.286,A -85,B 0,C 180,E1 -443.484,E2 -443.484} C_VEL
LIN {X 0,Y 608.45,Z 543.865,A -85,B 0,C 180,E1 -444.366,E2 -444.366} C_VEL
LIN {X 0,Y 608.432,Z 548.95,A -85,B 0,C 180,E1 -445.362,E2 -445.362} C_VEL
LIN {X 0,Y 608.449,Z 552.896,A -85,B 0,C 180,E1 -446.358,E2 -446.358} C_VEL
LIN {X 0,Y 608.425,Z 555.809,A -85,B 0,C 180,E1 -447.352,E2 -447.352} C_VEL
LIN {X 0,Y 608.444,Z 557.201,A -85,B 0,C 180,E1 -448.014,E2 -448.014} C_VEL
LIN {X 0,Y 608.438,Z 558.783,A -85,B 0,C 180,E1 -449.338,E2 -449.338} C_VEL
LIN {X 0,Y 608.434,Z 559,A -85,B 0,C 180,E1 -450,E2 -450} C_VEL
LIN {X 0,Y 608.448,Z 558.184,A -85,B 0,C 180,E1 -451.324,E2 -451.324} C_VEL
LIN {X 0,Y 608.444,Z 557.202,A -85,B 0,C 180,E1 -451.986,E2 -451.986} C_VEL
LIN {X 0,Y 608.425,Z 555.81,A -85,B 0,C 180,E1 -452.648,E2 -452.648} C_VEL
LIN {X 0,Y 608.449,Z 552.897,A -85,B 0,C 180,E1 -453.642,E2 -453.642} C_VEL
LIN {X 0,Y 608.432,Z 548.951,A -85,B 0,C 180,E1 -454.638,E2 -454.638} C_VEL
LIN {X 0,Y 608.437,Z 542.878,A -85,B 0,C 180,E1 -455.801,E2 -455.801} C_VEL
LIN {X 0,Y 608.462,Z 536.237,A -85,B 0,C 180,E1 -456.799,E2 -456.799} C_VEL
LIN {X 0,Y 608.455,Z 527.992,A -85,B 0,C 180,E1 -457.8,E2 -457.8} C_VEL
LIN {X 0,Y 608.472,Z 519.54,A -85,B 0,C 180,E1 -458.635,E2 -458.635} C_VEL
LIN {X 0,Y 608.481,Z 509.095,A -85,B 0,C 180,E1 -459.473,E2 -459.473} C_VEL
LIN {X 0,Y 608.499,Z 498.761,A -85,B 0,C 180,E1 -460.144,E2 -460.144} C_VEL
LIN {X 0,Y 608.472,Z 487.828,A -85,B 0,C 180,E1 -460.714,E2 -460.714} C_VEL
LIN {X 0,Y 608.494,Z 476.073,A -85,B 0,C 180,E1 -461.187,E2 -461.187} C_VEL
LIN {X 0,Y 608.549,Z 463.284,A -85,B 0,C 180,E1 -461.554,E2 -461.554} C_VEL
LIN {X 0,Y 608.444,Z 451.532,A -85,B 0,C 180,E1 -461.788,E2 -461.788} C_VEL
LIN {X 0,Y 608.434,Z 441.437,A -85,B 0,C 180,E1 -464.379,E2 -464.379} C_VEL
LIN {X 0,Y 608.445,Z 430.846,A -85,B 0,C 180,E1 -467.13,E2 -467.13} C_VEL
LIN {X 0,Y 608.454,Z 421.579,A -85,B 0,C 180,E1 -469.57,E2 -469.57} C_VEL
LIN {X 0,Y 608.461,Z 410.726,A -85,B 0,C 180,E1 -472.476,E2 -472.476} C_VEL
LIN {X 0,Y 608.435,Z 401.721,A -85,B 0,C 180,E1 -474.935,E2 -474.935} C_VEL
LIN {X 0,Y 608.444,Z 393.58,A -85,B 0,C 180,E1 -477.201,E2 -477.201} C_VEL
LIN {X 0,Y 608.476,Z 383.836,A -85,B 0,C 180,E1 -479.973,E2 -479.973} C_VEL
LIN {X 0,Y 608.481,Z 375.106,A -85,B 0,C 180,E1 -482.525,E2 -482.525} C_VEL
LIN {X 0,Y 608.555,Z 365.977,A -85,B 0,C 180,E1 -485.269,E2 -485.269} C_VEL
LIN {X 0,Y 608.485,Z 364.692,A -85,B 0,C 180,E1 -485.68,E2 -485.68} C_VEL
LIN {X 0,Y 608.46,Z 364.696,A -85,B 0,C 180,E1 -488.588,E2 -488.588} C_VEL
LIN {X 0,Y 608.465,Z 364.694,A -85,B 0,C 180,E1 -491.342,E2 -491.342} C_VEL
LIN {X 0,Y 608.456,Z 364.696,A -85,B 0,C 180,E1 -494.264,E2 -494.264} C_VEL
LIN {X 0,Y 608.442,Z 364.697,A -85,B 0,C 180,E1 -497.039,E2 -497.039} C_VEL
LIN {X 0,Y 608.448,Z 364.697,A -85,B 0,C 180,E1 -499.696,E2 -499.696} C_VEL
LIN {X 0,Y 608.467,Z 364.693,A -85,B 0,C 180,E1 -502.253,E2 -502.253} C_VEL
LIN {X 0,Y 608.484,Z 364.694,A -85,B 0,C 180,E1 -505.088,E2 -505.088} C_VEL
LIN {X 0,Y 608.462,Z 364.694,A -85,B 0,C 180,E1 -507.905,E2 -507.905} C_VEL
LIN {X 0,Y 608.458,Z 364.694,A -85,B 0,C 180,E1 -510.22,E2 -510.22} C_VEL
LIN {X 0,Y 608.481,Z 364.694,A -85,B 0,C 180,E1 -512.79,E2 -512.79} C_VEL
LIN {X 0,Y 608.475,Z 364.693,A -85,B 0,C 180,E1 -515.845,E2 -515.845} C_VEL
LIN {X 0,Y 608.463,Z 364.696,A -85,B 0,C 180,E1 -518.308,E2 -518.308} C_VEL
LIN {X 0,Y 608.471,Z 364.693,A -85,B 0,C 180,E1 -521.28,E2 -521.28} C_VEL
LIN {X 0,Y 608.459,Z 364.697,A -85,B 0,C 180,E1 -523.906,E2 -523.906} C_VEL
LIN {X 0,Y 608.459,Z 364.694,A -85,B 0,C 180,E1 -526.643,E2 -526.643} C_VEL
LIN {X 0,Y 608.468,Z 364.696,A -85,B 0,C 180,E1 -529.35,E2 -529.35} C_VEL
LIN {X 0,Y 608.466,Z 364.694,A -85,B 0,C 180,E1 -532.033,E2 -532.033} C_VEL
LIN {X 0,Y 608.458,Z 364.695,A -85,B 0,C 180,E1 -534.698,E2 -534.698} C_VEL
LIN {X 0,Y 608.47,Z 364.694,A -85,B 0,C 180,E1 -537.352,E2 -537.352} C_VEL
LIN {X 0,Y 608.463,Z 364.694,A -85,B 0,C 180,E1 -540,E2 -540} C_VEL
LIN {X 0,Y 608.478,Z 364.695,A -85,B 0,C 180,E1 -542.648,E2 -542.648} C_VEL
LIN {X 0,Y 608.459,Z 364.694,A -85,B 0,C 180,E1 -545.302,E2 -545.302} C_VEL
LIN {X 0,Y 608.468,Z 364.694,A -85,B 0,C 180,E1 -547.967,E2 -547.967} C_VEL
LIN {X 0,Y 608.46,Z 364.695,A -85,B 0,C 180,E1 -549.466,E2 -549.466} C_VEL
LIN {X 0,Y 607.772,Z 364.78,A -85,B 0,C 180,E1 -550.018,E2 -550.018} C_VEL
LIN {X 0,Y 604.913,Z 365.136,A -85,B 0,C 180,E1 -550.915,E2 -550.915} C_VEL
LIN {X 0,Y 602.513,Z 365.437,A -85,B 0,C 180,E1 -551.637,E2 -551.637} C_VEL
LIN {X 0,Y 601.487,Z 365.563,A -85,B 0,C 180,E1 -552.193,E2 -552.193} C_VEL
LIN {X 0,Y 601.405,Z 365.572,A -85,B 0,C 180,E1 -552.382,E2 -552.382} C_VEL
LIN {X 0,Y 601.421,Z 365.574,A -85,B 0,C 180,E1 -554.897,E2 -554.897} C_VEL
LIN {X 0,Y 601.427,Z 365.572,A -85,B 0,C 180,E1 -556.986,E2 -556.986} C_VEL
LIN {X 0,Y 601.402,Z 365.573,A -85,B 0,C 180,E1 -559.81,E2 -559.81} C_VEL
LIN {X 0,Y 601.407,Z 365.576,A -85,B 0,C 180,E1 -562.606,E2 -562.606} C_VEL
LIN {X 0,Y 601.396,Z 365.577,A -85,B 0,C 180,E1 -564.879,E2 -564.879} C_VEL
LIN {X 0,Y 601.417,Z 365.572,A -85,B 0,C 180,E1 -567.365,E2 -567.365} C_VEL
LIN {X 0,Y 601.42,Z 365.572,A -85,B 0,C 180,E1 -570.149,E2 -570.149} C_VEL
LIN {X 0,Y 601.417,Z 365.573,A -85,B 0,C 180,E1 -572.717,E2 -572.717} C_VEL
LIN {X 0,Y 601.414,Z 365.572,A -85,B 0,C 180,E1 -575.116,E2 -575.116} C_VEL
LIN {X 0,Y 601.431,Z 365.57,A -85,B 0,C 180,E1 -577.42,E2 -577.42} C_VEL
LIN {X 0,Y 601.407,Z 365.573,A -85,B 0,C 180,E1 -579.996,E2 -579.996} C_VEL
LIN {X 0,Y 601.404,Z 365.575,A -85,B 0,C 180,E1 -582.671,E2 -582.671} C_VEL
LIN {X 0,Y 601.422,Z 365.571,A -85,B 0,C 180,E1 -585.483,E2 -585.483} C_VEL
LIN {X 0,Y 601.426,Z 365.571,A -85,B 0,C 180,E1 -588.407,E2 -588.407} C_VEL
LIN {X 0,Y 601.432,Z 365.569,A -85,B 0,C 180,E1 -590.876,E2 -590.876} C_VEL
LIN {X 0,Y 601.441,Z 365.57,A -85,B 0,C 180,E1 -593.735,E2 -593.735} C_VEL
LIN {X 0,Y 601.429,Z 365.571,A -85,B 0,C 180,E1 -596.688,E2 -596.688} C_VEL
LIN {X 0,Y 601.431,Z 365.572,A -85,B 0,C 180,E1 -599.06,E2 -599.06} C_VEL
LIN {X 0,Y 601.432,Z 365.573,A -85,B 0,C 180,E1 -601.374,E2 -601.374} C_VEL
LIN {X 0,Y 601.422,Z 365.571,A -85,B 0,C 180,E1 -604.132,E2 -604.132} C_VEL
LIN {X 0,Y 601.423,Z 365.571,A -85,B 0,C 180,E1 -606.59,E2 -606.59} C_VEL
LIN {X 0,Y 601.426,Z 365.571,A -85,B 0,C 180,E1 -609.479,E2 -609.479} C_VEL
LIN {X 0,Y 601.395,Z 365.576,A -85,B 0,C 180,E1 -612.312,E2 -612.312} C_VEL
LIN {X 0,Y 601.415,Z 365.573,A -85,B 0,C 180,E1 -614.409,E2 -614.409} C_VEL
LIN {X 0,Y 601.415,Z 365.572,A -85,B 0,C 180,E1 -617.172,E2 -617.172} C_VEL
LIN {X 0,Y 601.438,Z 365.57,A -85,B 0,C 180,E1 -619.905,E2 -619.905} C_VEL
LIN {X 0,Y 601.41,Z 365.573,A -85,B 0,C 180,E1 -622.615,E2 -622.615} C_VEL
LIN {X 0,Y 601.417,Z 365.572,A -85,B 0,C 180,E1 -625.308,E2 -625.308} C_VEL
LIN {X 0,Y 601.406,Z 365.574,A -85,B 0,C 180,E1 -626.651,E2 -626.651} C_VEL
LIN {X 0,Y 601.363,Z 365.921,A -85,B 0,C 180,E1 -627.321,E2 -627.321} C_VEL
LIN {X 0,Y 601.384,Z 369.124,A -85,B 0,C 180,E1 -630,E2 -630} C_VEL
LIN {X 0,Y 601.312,Z 372.268,A -85,B 0,C 180,E1 -632.68,E2 -632.68} C_VEL
LIN {X 0,Y 601.365,Z 375.654,A -85,B 0,C 180,E1 -635.365,E2 -635.365} C_VEL
LIN {X 0,Y 601.348,Z 379.154,A -85,B 0,C 180,E1 -638.062,E2 -638.062} C_VEL
LIN {X 0,Y 601.329,Z 383,A -85,B 0,C 180,E1 -640.963,E2 -640.963} C_VEL
LIN {X 0,Y 601.334,Z 386.449,A -85,B 0,C 180,E1 -643.518,E2 -643.518} C_VEL
LIN {X 0,Y 601.322,Z 390.662,A -85,B 0,C 180,E1 -646.587,E2 -646.587} C_VEL
LIN {X 0,Y 601.307,Z 394.162,A -85,B 0,C 180,E1 -649.102,E2 -649.102} C_VEL
LIN {X 0,Y 601.348,Z 395.685,A -85,B 0,C 180,E1 -650.19,E2 -650.19} C_VEL
LIN {X 0,Y 601.587,Z 407.002,A -85,B 0,C 180,E1 -650.449,E2 -650.449} C_VEL
LIN {X 0,Y 601.538,Z 420.346,A -85,B 0,C 180,E1 -650.887,E2 -650.887} C_VEL
LIN {X 0,Y 601.525,Z 432.115,A -85,B 0,C 180,E1 -651.414,E2 -651.414} C_VEL
LIN {X 0,Y 601.486,Z 443.062,A -85,B 0,C 180,E1 -652.045,E2 -652.045} C_VEL
LIN {X 0,Y 601.457,Z 454.324,A -85,B 0,C 180,E1 -652.862,E2 -652.862} C_VEL
LIN {X 0,Y 601.426,Z 462.55,A -85,B 0,C 180,E1 -653.592,E2 -653.592} C_VEL
LIN {X 0,Y 601.408,Z 471.43,A -85,B 0,C 180,E1 -654.548,E2 -654.548} C_VEL
LIN {X 0,Y 601.357,Z 479.406,A -85,B 0,C 180,E1 -655.621,E2 -655.621} C_VEL
LIN {X 0,Y 601.355,Z 486.001,A -85,B 0,C 180,E1 -656.74,E2 -656.74} C_VEL
LIN {X 0,Y 601.354,Z 491.11,A -85,B 0,C 180,E1 -657.87,E2 -657.87} C_VEL
LIN {X 0,Y 601.342,Z 494.198,A -85,B 0,C 180,E1 -658.772,E2 -658.772} C_VEL
LIN {X 0,Y 601.344,Z 495.885,A -85,B 0,C 180,E1 -659.397,E2 -659.397} C_VEL
LIN {X 0,Y 601.347,Z 497.419,A -85,B 0,C 180,E1 -660.168,E2 -660.168} C_VEL
LIN {X 0,Y 601.33,Z 498.829,A -85,B 0,C 180,E1 -661.44,E2 -661.44} C_VEL
LIN {X 0,Y 601.325,Z 498.794,A -85,B 0,C 180,E1 -662.7,E2 -662.7} C_VEL
LIN {X 0,Y 601.324,Z 497.423,A -85,B 0,C 180,E1 -663.92,E2 -663.92} C_VEL
LIN {X 0,Y 601.32,Z 494.817,A -85,B 0,C 180,E1 -665.101,E2 -665.101} C_VEL
LIN {X 0,Y 601.338,Z 490.991,A -85,B 0,C 180,E1 -666.252,E2 -666.252} C_VEL
LIN {X 0,Y 601.365,Z 485.606,A -85,B 0,C 180,E1 -667.423,E2 -667.423} C_VEL
LIN {X 0,Y 601.372,Z 478.584,A -85,B 0,C 180,E1 -668.593,E2 -668.593} C_VEL
LIN {X 0,Y 601.402,Z 471.525,A -85,B 0,C 180,E1 -669.531,E2 -669.531} C_VEL
LIN {X 0,Y 601.4,Z 463.376,A -85,B 0,C 180,E1 -670.419,E2 -670.419} C_VEL
LIN {X 0,Y 601.452,Z 453.235,A -85,B 0,C 180,E1 -671.315,E2 -671.315} C_VEL
LIN {X 0,Y 601.446,Z 442.227,A -85,B 0,C 180,E1 -672.1,E2 -672.1} C_VEL
LIN {X 0,Y 601.457,Z 431.186,A -85,B 0,C 180,E1 -672.722,E2 -672.722} C_VEL
LIN {X 0,Y 601.489,Z 419.547,A -85,B 0,C 180,E1 -673.234,E2 -673.234} C_VEL
LIN {X 0,Y 601.562,Z 406.939,A -85,B 0,C 180,E1 -673.643,E2 -673.643} C_VEL
LIN {X 0,Y 601.42,Z 396.83,A -85,B 0,C 180,E1 -673.874,E2 -673.874} C_VEL
LIN {X 0,Y 601.3,Z 395.655,A -85,B 0,C 180,E1 -673.923,E2 -673.923} C_VEL
LIN {X 0,Y 601.295,Z 392.137,A -85,B 0,C 180,E1 -676.44,E2 -676.44} C_VEL
LIN {X 0,Y 601.287,Z 387.997,A -85,B 0,C 180,E1 -679.44,E2 -679.44} C_VEL
LIN {X 0,Y 601.298,Z 384.891,A -85,B 0,C 180,E1 -681.723,E2 -681.723} C_VEL
LIN {X 0,Y 601.296,Z 381.519,A -85,B 0,C 180,E1 -684.239,E2 -684.239} C_VEL
LIN {X 0,Y 601.331,Z 378.302,A -85,B 0,C 180,E1 -686.68,E2 -686.68} C_VEL
LIN {X 0,Y 601.339,Z 375.236,A -85,B 0,C 180,E1 -689.053,E2 -689.053} C_VEL
LIN {X 0,Y 601.347,Z 372.35,A -85,B 0,C 180,E1 -691.369,E2 -691.369} C_VEL
LIN {X 0,Y 601.385,Z 369.138,A -85,B 0,C 180,E1 -694.136,E2 -694.136} C_VEL
LIN {X 0,Y 601.382,Z 366.206,A -85,B 0,C 180,E1 -696.588,E2 -696.588} C_VEL
LIN {X 0,Y 601.409,Z 365.575,A -85,B 0,C 180,E1 -697.394,E2 -697.394} C_VEL
LIN {X 0,Y 601.401,Z 365.573,A -85,B 0,C 180,E1 -700.19,E2 -700.19} C_VEL
LIN {X 0,Y 601.428,Z 365.57,A -85,B 0,C 180,E1 -703.014,E2 -703.014} C_VEL
LIN {X 0,Y 601.415,Z 365.574,A -85,B 0,C 180,E1 -705.907,E2 -705.907} C_VEL
LIN {X 0,Y 601.43,Z 365.57,A -85,B 0,C 180,E1 -708.542,E2 -708.542} C_VEL
LIN {X 0,Y 601.437,Z 365.568,A -85,B 0,C 180,E1 -711.262,E2 -711.262} C_VEL
LIN {X 0,Y 601.406,Z 365.573,A -85,B 0,C 180,E1 -713.963,E2 -713.963} C_VEL
LIN {X 0,Y 601.431,Z 365.572,A -85,B 0,C 180,E1 -716.65,E2 -716.65} C_VEL
LIN {X 0,Y 601.444,Z 365.569,A -85,B 0,C 180,E1 -719.33,E2 -719.33} C_VEL
LIN {X 0,Y 601.41,Z 365.572,A -85,B 0,C 180,E1 -722.009,E2 -722.009} C_VEL
LIN {X 0,Y 601.415,Z 365.571,A -85,B 0,C 180,E1 -724.692,E2 -724.692} C_VEL
LIN {X 0,Y 601.449,Z 365.568,A -85,B 0,C 180,E1 -727.385,E2 -727.385} C_VEL
LIN {X 0,Y 601.432,Z 365.572,A -85,B 0,C 180,E1 -730.095,E2 -730.095} C_VEL
LIN {X 0,Y 601.423,Z 365.57,A -85,B 0,C 180,E1 -732.828,E2 -732.828} C_VEL
LIN {X 0,Y 601.407,Z 365.572,A -85,B 0,C 180,E1 -735.591,E2 -735.591} C_VEL
LIN {X 0,Y 601.395,Z 365.574,A -85,B 0,C 180,E1 -737.688,E2 -737.688} C_VEL
LIN {X 0,Y 601.426,Z 365.57,A -85,B 0,C 180,E1 -740.522,E2 -740.522} C_VEL
LIN {X 0,Y 601.415,Z 365.574,A -85,B 0,C 180,E1 -743.411,E2 -743.411} C_VEL
LIN {X 0,Y 601.404,Z 365.572,A -85,B 0,C 180,E1 -746.364,E2 -746.364} C_VEL
LIN {X 0,Y 601.441,Z 365.568,A -85,B 0,C 180,E1 -748.791,E2 -748.791} C_VEL
LIN {X 0,Y 601.398,Z 365.576,A -85,B 0,C 180,E1 -751.727,E2 -751.727} C_VEL
LIN {X 0,Y 601.417,Z 365.573,A -85,B 0,C 180,E1 -754.119,E2 -754.119} C_VEL
LIN {X 0,Y 601.395,Z 365.577,A -85,B 0,C 180,E1 -756.584,E2 -756.584} C_VEL
LIN {X 0,Y 601.435,Z 365.572,A -85,B 0,C 180,E1 -759.125,E2 -759.125} C_VEL
LIN {X 0,Y 601.42,Z 365.572,A -85,B 0,C 180,E1 -761.766,E2 -761.766} C_VEL
LIN {X 0,Y 601.422,Z 365.57,A -85,B 0,C 180,E1 -764.536,E2 -764.536} C_VEL
LIN {X 0,Y 601.412,Z 365.574,A -85,B 0,C 180,E1 -767.41,E2 -767.41} C_VEL
LIN {X 0,Y 601.441,Z 365.568,A -85,B 0,C 180,E1 -770.464,E2 -770.464} C_VEL
LIN {X 0,Y 601.403,Z 365.575,A -85,B 0,C 180,E1 -773.418,E2 -773.418} C_VEL
LIN {X 0,Y 601.472,Z 365.686,A -85,B 0,C 180,E1 -774.162,E2 -774.162} C_VEL
LIN {X 0,Y 601.578,Z 373.918,A -85,B 0,C 180,E1 -776.696,E2 -776.696} C_VEL
LIN {X 0,Y 601.495,Z 381.862,A -85,B 0,C 180,E1 -779.063,E2 -779.063} C_VEL
LIN {X 0,Y 601.453,Z 389.805,A -85,B 0,C 180,E1 -781.375,E2 -781.375} C_VEL
LIN {X 0,Y 601.483,Z 400.396,A -85,B 0,C 180,E1 -784.385,E2 -784.385} C_VEL
LIN {X 0,Y 601.411,Z 409.663,A -85,B 0,C 180,E1 -786.954,E2 -786.954} C_VEL
LIN {X 0,Y 601.432,Z 418.93,A -85,B 0,C 180,E1 -789.478,E2 -789.478} C_VEL
LIN {X 0,Y 601.404,Z 429.521,A -85,B 0,C 180,E1 -792.312,E2 -792.312} C_VEL
LIN {X 0,Y 601.368,Z 440.112,A -85,B 0,C 180,E1 -795.102,E2 -795.102} C_VEL
LIN {X 0,Y 601.35,Z 449.379,A -85,B 0,C 180,E1 -797.514,E2 -797.514} C_VEL
LIN {X 0,Y 601.383,Z 451.53,A -85,B 0,C 180,E1 -798.071,E2 -798.071} C_VEL
LIN {X 0,Y 601.6,Z 465.936,A -85,B 0,C 180,E1 -798.374,E2 -798.374} C_VEL
LIN {X 0,Y 601.514,Z 478.263,A -85,B 0,C 180,E1 -798.762,E2 -798.762} C_VEL
LIN {X 0,Y 601.485,Z 490.923,A -85,B 0,C 180,E1 -799.31,E2 -799.31} C_VEL
LIN {X 0,Y 601.474,Z 501.58,A -85,B 0,C 180,E1 -799.906,E2 -799.906} C_VEL
LIN {X 0,Y 601.449,Z 512.475,A -85,B 0,C 180,E1 -800.669,E2 -800.669} C_VEL
LIN {X 0,Y 601.429,Z 523.112,A -85,B 0,C 180,E1 -801.601,E2 -801.601} C_VEL
LIN {X 0,Y 601.418,Z 530.96,A -85,B 0,C 180,E1 -802.446,E2 -802.446} C_VEL
LIN {X 0,Y 601.37,Z 538.224,A -85,B 0,C 180,E1 -803.398,E2 -803.398} C_VEL
LIN {X 0,Y 601.372,Z 543.866,A -85,B 0,C 180,E1 -804.299,E2 -804.299} C_VEL
LIN {X 0,Y 601.336,Z 548.95,A -85,B 0,C 180,E1 -805.307,E2 -805.307} C_VEL
LIN {X 0,Y 601.368,Z 552.896,A -85,B 0,C 180,E1 -806.315,E2 -806.315} C_VEL
LIN {X 0,Y 601.325,Z 555.809,A -85,B 0,C 180,E1 -807.32,E2 -807.32} C_VEL
LIN {X 0,Y 601.343,Z 557.201,A -85,B 0,C 180,E1 -807.991,E2 -807.991} C_VEL
LIN {X 0,Y 601.339,Z 558.783,A -85,B 0,C 180,E1 -809.33,E2 -809.33} C_VEL
LIN {X 0,Y 601.335,Z 559,A -85,B 0,C 180,E1 -810,E2 -810} C_VEL
LIN {X 0,Y 601.347,Z 558.184,A -85,B 0,C 180,E1 -811.339,E2 -811.339} C_VEL
LIN {X 0,Y 601.343,Z 557.202,A -85,B 0,C 180,E1 -812.009,E2 -812.009} C_VEL
LIN {X 0,Y 601.325,Z 555.81,A -85,B 0,C 180,E1 -812.679,E2 -812.679} C_VEL
LIN {X 0,Y 601.368,Z 552.897,A -85,B 0,C 180,E1 -813.685,E2 -813.685} C_VEL
LIN {X 0,Y 601.336,Z 548.951,A -85,B 0,C 180,E1 -814.692,E2 -814.692} C_VEL
LIN {X 0,Y 601.372,Z 542.878,A -85,B 0,C 180,E1 -815.869,E2 -815.869} C_VEL
LIN {X 0,Y 601.381,Z 536.237,A -85,B 0,C 180,E1 -816.879,E2 -816.879} C_VEL
LIN {X 0,Y 601.4,Z 527.992,A -85,B 0,C 180,E1 -817.892,E2 -817.892} C_VEL
LIN {X 0,Y 601.436,Z 519.54,A -85,B 0,C 180,E1 -818.737,E2 -818.737} C_VEL
LIN {X 0,Y 601.451,Z 509.096,A -85,B 0,C 180,E1 -819.585,E2 -819.585} C_VEL
LIN {X 0,Y 601.489,Z 498.762,A -85,B 0,C 180,E1 -820.264,E2 -820.264} C_VEL
LIN {X 0,Y 601.49,Z 487.147,A -85,B 0,C 180,E1 -820.872,E2 -820.872} C_VEL
LIN {X 0,Y 601.527,Z 474.33,A -85,B 0,C 180,E1 -821.376,E2 -821.376} C_VEL
LIN {X 0,Y 601.618,Z 461.456,A -85,B 0,C 180,E1 -821.732,E2 -821.732} C_VEL
LIN {X 0,Y 601.383,Z 451.532,A -85,B 0,C 180,E1 -821.929,E2 -821.929} C_VEL
LIN {X 0,Y 601.383,Z 441.437,A -85,B 0,C 180,E1 -824.551,E2 -824.551} C_VEL
LIN {X 0,Y 601.39,Z 430.846,A -85,B 0,C 180,E1 -827.337,E2 -827.337} C_VEL
LIN {X 0,Y 601.428,Z 420.255,A -85,B 0,C 180,E1 -830.164,E2 -830.164} C_VEL
LIN {X 0,Y 601.428,Z 410.988,A -85,B 0,C 180,E1 -832.682,E2 -832.682} C_VEL
LIN {X 0,Y 601.433,Z 401.721,A -85,B 0,C 180,E1 -835.246,E2 -835.246} C_VEL
LIN {X 0,Y 601.499,Z 392.454,A -85,B 0,C 180,E1 -837.863,E2 -837.863} C_VEL
LIN {X 0,Y 601.469,Z 383.187,A -85,B 0,C 180,E1 -840.549,E2 -840.549} C_VEL
LIN {X 0,Y 601.515,Z 375.837,A -85,B 0,C 180,E1 -842.729,E2 -842.729} C_VEL
LIN {X 0,Y 601.587,Z 367.918,A -85,B 0,C 180,E1 -845.137,E2 -845.137} C_VEL
LIN {X 0,Y 601.447,Z 365.57,A -85,B 0,C 180,E1 -845.93,E2 -845.93} C_VEL
LIN {X 0,Y 601.427,Z 365.573,A -85,B 0,C 180,E1 -848.47,E2 -848.47} C_VEL
LIN {X 0,Y 601.423,Z 365.572,A -85,B 0,C 180,E1 -851.593,E2 -851.593} C_VEL
LIN {X 0,Y 601.419,Z 365.571,A -85,B 0,C 180,E1 -854.534,E2 -854.534} C_VEL
LIN {X 0,Y 601.408,Z 365.575,A -85,B 0,C 180,E1 -857.408,E2 -857.408} C_VEL
LIN {X 0,Y 601.432,Z 365.571,A -85,B 0,C 180,E1 -860.464,E2 -860.464} C_VEL
LIN {X 0,Y 601.413,Z 365.572,A -85,B 0,C 180,E1 -863.418,E2 -863.418} C_VEL
LIN {X 0,Y 601.428,Z 365.572,A -85,B 0,C 180,E1 -866.063,E2 -866.063} C_VEL
LIN {X 0,Y 601.435,Z 365.571,A -85,B 0,C 180,E1 -868.541,E2 -868.541} C_VEL
LIN {X 0,Y 601.438,Z 365.569,A -85,B 0,C 180,E1 -871.373,E2 -871.373} C_VEL
LIN {X 0,Y 601.402,Z 365.574,A -85,B 0,C 180,E1 -873.636,E2 -873.636} C_VEL
LIN {X 0,Y 601.417,Z 365.572,A -85,B 0,C 180,E1 -876.59,E2 -876.59} C_VEL
LIN {X 0,Y 601.431,Z 365.573,A -85,B 0,C 180,E1 -879.478,E2 -879.478} C_VEL
LIN {X 0,Y 601.395,Z 365.574,A -85,B 0,C 180,E1 -882.312,E2 -882.312} C_VEL
LIN {X 0,Y 601.411,Z 365.572,A -85,B 0,C 180,E1 -884.409,E2 -884.409} C_VEL
LIN {X 0,Y 601.414,Z 365.575,A -85,B 0,C 180,E1 -887.172,E2 -887.172} C_VEL
LIN {X 0,Y 601.426,Z 365.57,A -85,B 0,C 180,E1 -889.905,E2 -889.905} C_VEL
LIN {X 0,Y 601.448,Z 365.57,A -85,B 0,C 180,E1 -892.615,E2 -892.615} C_VEL
LIN {X 0,Y 601.413,Z 365.572,A -85,B 0,C 180,E1 -895.308,E2 -895.308} C_VEL
LIN {X 0,Y 601.42,Z 365.572,A -85,B 0,C 180,E1 -897.991,E2 -897.991} C_VEL
LIN {X 0,Y 601.455,Z 365.568,A -85,B 0,C 180,E1 -900.67,E2 -900.67} C_VEL
LIN {X 0,Y 601.428,Z 365.57,A -85,B 0,C 180,E1 -903.35,E2 -903.35} C_VEL
LIN {X 0,Y 601.413,Z 365.575,A -85,B 0,C 180,E1 -906.037,E2 -906.037} C_VEL
LIN {X 0,Y 601.438,Z 365.569,A -85,B 0,C 180,E1 -908.738,E2 -908.738} C_VEL
LIN {X 0,Y 601.429,Z 365.572,A -85,B 0,C 180,E1 -911.458,E2 -911.458} C_VEL
LIN {X 0,Y 601.405,Z 365.572,A -85,B 0,C 180,E1 -912.382,E2 -912.382} C_VEL
LIN {X 0,Y 600.742,Z 365.657,A -85,B 0,C 180,E1 -912.941,E2 -912.941} C_VEL
LIN {X 0,Y 597.89,Z 366.013,A -85,B 0,C 180,E1 -913.849,E2 -913.849} C_VEL
LIN {X 0,Y 595.477,Z 366.313,A -85,B 0,C 180,E1 -914.579,E2 -914.579} C_VEL
LIN {X 0,Y 594.439,Z 366.441,A -85,B 0,C 180,E1 -915.143,E2 -915.143} C_VEL
LIN {X 0,Y 594.354,Z 366.451,A -85,B 0,C 180,E1 -915.333,E2 -915.333} C_VEL
LIN {X 0,Y 594.373,Z 366.449,A -85,B 0,C 180,E1 -917.905,E2 -917.905} C_VEL
LIN {X 0,Y 594.382,Z 366.448,A -85,B 0,C 180,E1 -920.92,E2 -920.92} C_VEL
LIN {X 0,Y 594.387,Z 366.45,A -85,B 0,C 180,E1 -923.704,E2 -923.704} C_VEL
LIN {X 0,Y 594.385,Z 366.448,A -85,B 0,C 180,E1 -926.7,E2 -926.7} C_VEL
LIN {X 0,Y 594.378,Z 366.449,A -85,B 0,C 180,E1 -928.999,E2 -928.999} C_VEL
LIN {X 0,Y 594.385,Z 366.449,A -85,B 0,C 180,E1 -931.646,E2 -931.646} C_VEL
LIN {X 0,Y 594.396,Z 366.447,A -85,B 0,C 180,E1 -934.579,E2 -934.579} C_VEL
LIN {X 0,Y 594.384,Z 366.45,A -85,B 0,C 180,E1 -937.087,E2 -937.087} C_VEL
LIN {X 0,Y 594.37,Z 366.449,A -85,B 0,C 180,E1 -939.775,E2 -939.775} C_VEL
LIN {X 0,Y 594.363,Z 366.452,A -85,B 0,C 180,E1 -942.376,E2 -942.376} C_VEL
LIN {X 0,Y 594.359,Z 366.45,A -85,B 0,C 180,E1 -945.192,E2 -945.192} C_VEL
LIN {X 0,Y 594.364,Z 366.45,A -85,B 0,C 180,E1 -947.625,E2 -947.625} C_VEL
LIN {X 0,Y 594.39,Z 366.449,A -85,B 0,C 180,E1 -950.322,E2 -950.322} C_VEL
LIN {X 0,Y 594.381,Z 366.448,A -85,B 0,C 180,E1 -952.914,E2 -952.914} C_VEL
LIN {X 0,Y 594.382,Z 366.451,A -85,B 0,C 180,E1 -955.862,E2 -955.862} C_VEL
LIN {X 0,Y 594.391,Z 366.447,A -85,B 0,C 180,E1 -958.652,E2 -958.652} C_VEL
LIN {X 0,Y 594.384,Z 366.448,A -85,B 0,C 180,E1 -961.043,E2 -961.043} C_VEL
LIN {X 0,Y 594.382,Z 366.448,A -85,B 0,C 180,E1 -964.057,E2 -964.057} C_VEL
LIN {X 0,Y 594.394,Z 366.446,A -85,B 0,C 180,E1 -966.297,E2 -966.297} C_VEL
LIN {X 0,Y 594.401,Z 366.447,A -85,B 0,C 180,E1 -969.225,E2 -969.225} C_VEL
LIN {X 0,Y 594.354,Z 366.452,A -85,B 0,C 180,E1 -972.096,E2 -972.096} C_VEL
LIN {X 0,Y 594.369,Z 366.45,A -85,B 0,C 180,E1 -974.22,E2 -974.22} C_VEL
LIN {X 0,Y 594.389,Z 366.447,A -85,B 0,C 180,E1 -976.322,E2 -976.322} C_VEL
LIN {X 0,Y 594.375,Z 366.452,A -85,B 0,C 180,E1 -979.095,E2 -979.095} C_VEL
LIN {X 0,Y 594.419,Z 366.443,A -85,B 0,C 180,E1 -981.844,E2 -981.844} C_VEL
LIN {X 0,Y 594.396,Z 366.449,A -85,B 0,C 180,E1 -984.573,E2 -984.573} C_VEL
LIN {X 0,Y 594.288,Z 366.498,A -85,B 0,C 180,E1 -987.289,E2 -987.289} C_VEL
LIN {X 0,Y 594.329,Z 369.714,A -85,B 0,C 180,E1 -990,E2 -990} C_VEL
LIN {X 0,Y 594.235,Z 372.874,A -85,B 0,C 180,E1 -992.712,E2 -992.712} C_VEL
LIN {X 0,Y 594.278,Z 376.171,A -85,B 0,C 180,E1 -995.429,E2 -995.429} C_VEL
LIN {X 0,Y 594.271,Z 379.673,A -85,B 0,C 180,E1 -998.159,E2 -998.159} C_VEL
LIN {X 0,Y 594.251,Z 383.401,A -85,B 0,C 180,E1 -1001.003,E2 -1001.003} C_VEL
LIN {X 0,Y 594.253,Z 386.978,A -85,B 0,C 180,E1 -1003.682,E2 -1003.682} C_VEL
LIN {X 0,Y 594.237,Z 391.03,A -85,B 0,C 180,E1 -1006.667,E2 -1006.667} C_VEL
LIN {X 0,Y 594.206,Z 394.708,A -85,B 0,C 180,E1 -1009.34,E2 -1009.34} C_VEL
LIN {X 0,Y 594.22,Z 395.673,A -85,B 0,C 180,E1 -1010.036,E2 -1010.036} C_VEL
LIN {X 0,Y 594.651,Z 399.7,A -85,B 0,C 180,E1 -1010.134,E2 -1010.134} C_VEL
LIN {X 0,Y 594.614,Z 411.799,A -85,B 0,C 180,E1 -1010.451,E2 -1010.451} C_VEL
LIN {X 0,Y 594.555,Z 424.015,A -85,B 0,C 180,E1 -1010.906,E2 -1010.906} C_VEL
LIN {X 0,Y 594.504,Z 435.977,A -85,B 0,C 180,E1 -1011.498,E2 -1011.498} C_VEL
LIN {X 0,Y 594.466,Z 446.209,A -85,B 0,C 180,E1 -1012.138,E2 -1012.138} C_VEL
LIN {X 0,Y 594.398,Z 456.853,A -85,B 0,C 180,E1 -1012.966,E2 -1012.966} C_VEL
LIN {X 0,Y 594.34,Z 466.448,A -85,B 0,C 180,E1 -1013.891,E2 -1013.891} C_VEL
LIN {X 0,Y 594.322,Z 474.321,A -85,B 0,C 180,E1 -1014.821,E2 -1014.821} C_VEL
LIN {X 0,Y 594.296,Z 481.939,A -85,B 0,C 180,E1 -1015.947,E2 -1015.947} C_VEL
LIN {X 0,Y 594.276,Z 487.972,A -85,B 0,C 180,E1 -1017.084,E2 -1017.084} C_VEL
LIN {X 0,Y 594.245,Z 492.614,A -85,B 0,C 180,E1 -1018.233,E2 -1018.233} C_VEL
LIN {X 0,Y 594.255,Z 494.954,A -85,B 0,C 180,E1 -1019.005,E2 -1019.005} C_VEL
LIN {X 0,Y 594.242,Z 497.676,A -85,B 0,C 180,E1 -1020.304,E2 -1020.304} C_VEL
LIN {X 0,Y 594.227,Z 498.908,A -85,B 0,C 180,E1 -1021.618,E2 -1021.618} C_VEL
LIN {X 0,Y 594.245,Z 498.622,A -85,B 0,C 180,E1 -1022.958,E2 -1022.958} C_VEL
LIN {X 0,Y 594.245,Z 497.135,A -85,B 0,C 180,E1 -1024.119,E2 -1024.119} C_VEL
LIN {X 0,Y 594.247,Z 494.017,A -85,B 0,C 180,E1 -1025.415,E2 -1025.415} C_VEL
LIN {X 0,Y 594.27,Z 490.312,A -85,B 0,C 180,E1 -1026.468,E2 -1026.468} C_VEL
LIN {X 0,Y 594.262,Z 485.052,A -85,B 0,C 180,E1 -1027.592,E2 -1027.592} C_VEL
LIN {X 0,Y 594.308,Z 478.43,A -85,B 0,C 180,E1 -1028.695,E2 -1028.695} C_VEL
LIN {X 0,Y 594.332,Z 471.016,A -85,B 0,C 180,E1 -1029.683,E2 -1029.683} C_VEL
LIN {X 0,Y 594.374,Z 461.551,A -85,B 0,C 180,E1 -1030.695,E2 -1030.695} C_VEL
LIN {X 0,Y 594.435,Z 451.605,A -85,B 0,C 180,E1 -1031.557,E2 -1031.557} C_VEL
LIN {X 0,Y 594.437,Z 441.104,A -85,B 0,C 180,E1 -1032.289,E2 -1032.289} C_VEL
LIN {X 0,Y 594.455,Z 428.904,A -85,B 0,C 180,E1 -1032.962,E2 -1032.962} C_VEL
LIN {X 0,Y 594.522,Z 417.442,A -85,B 0,C 180,E1 -1033.448,E2 -1033.448} C_VEL
LIN {X 0,Y 594.626,Z 404.801,A -85,B 0,C 180,E1 -1033.838,E2 -1033.838} C_VEL
LIN {X 0,Y 594.487,Z 397.513,A -85,B 0,C 180,E1 -1034.001,E2 -1034.001} C_VEL
LIN {X 0,Y 594.203,Z 395.66,A -85,B 0,C 180,E1 -1034.063,E2 -1034.063} C_VEL
LIN {X 0,Y 594.202,Z 392.042,A -85,B 0,C 180,E1 -1036.685,E2 -1036.685} C_VEL
LIN {X 0,Y 594.209,Z 388.314,A -85,B 0,C 180,E1 -1039.419,E2 -1039.419} C_VEL
LIN {X 0,Y 594.208,Z 384.297,A -85,B 0,C 180,E1 -1042.413,E2 -1042.413} C_VEL
LIN {X 0,Y 594.218,Z 381.288,A -85,B 0,C 180,E1 -1044.693,E2 -1044.693} C_VEL
LIN {X 0,Y 594.253,Z 378.157,A -85,B 0,C 180,E1 -1047.106,E2 -1047.106} C_VEL
LIN {X 0,Y 594.245,Z 374.869,A -85,B 0,C 180,E1 -1049.694,E2 -1049.694} C_VEL
LIN {X 0,Y 594.308,Z 371.662,A -85,B 0,C 180,E1 -1052.536,E2 -1052.536} C_VEL
LIN {X 0,Y 594.322,Z 368.973,A -85,B 0,C 180,E1 -1054.804,E2 -1054.804} C_VEL
LIN {X 0,Y 594.316,Z 366.459,A -85,B 0,C 180,E1 -1057.031,E2 -1057.031} C_VEL
LIN {X 0,Y 594.407,Z 366.444,A -85,B 0,C 180,E1 -1059.224,E2 -1059.224} C_VEL
LIN {X 0,Y 594.376,Z 366.451,A -85,B 0,C 180,E1 -1062.096,E2 -1062.096} C_VEL
LIN {X 0,Y 594.36,Z 366.45,A -85,B 0,C 180,E1 -1064.219,E2 -1064.219} C_VEL
LIN {X 0,Y 594.375,Z 366.448,A -85,B 0,C 180,E1 -1066.321,E2 -1066.321} C_VEL
LIN {X 0,Y 594.378,Z 366.448,A -85,B 0,C 180,E1 -1069.095,E2 -1069.095} C_VEL
LIN {X 0,Y 594.41,Z 366.447,A -85,B 0,C 180,E1 -1071.843,E2 -1071.843} C_VEL
LIN {X 0,Y 594.391,Z 366.447,A -85,B 0,C 180,E1 -1074.572,E2 -1074.572} C_VEL
LIN {X 0,Y 594.405,Z 366.444,A -85,B 0,C 180,E1 -1077.289,E2 -1077.289} C_VEL
LIN {X 0,Y 594.402,Z 366.445,A -85,B 0,C 180,E1 -1080,E2 -1080} C_VEL
LIN {X 0,Y 594.405,Z 366.448,A -85,B 0,C 180,E1 -1082.711,E2 -1082.711} C_VEL
LIN {X 0,Y 594.39,Z 366.447,A -85,B 0,C 180,E1 -1085.428,E2 -1085.428} C_VEL
LIN {X 0,Y 594.407,Z 366.444,A -85,B 0,C 180,E1 -1088.157,E2 -1088.157} C_VEL
LIN {X 0,Y 594.388,Z 366.448,A -85,B 0,C 180,E1 -1091.077,E2 -1091.077} C_VEL
LIN {X 0,Y 594.378,Z 366.451,A -85,B 0,C 180,E1 -1093.679,E2 -1093.679} C_VEL
LIN {X 0,Y 594.393,Z 366.445,A -85,B 0,C 180,E1 -1096.722,E2 -1096.722} C_VEL
LIN {X 0,Y 594.363,Z 366.45,A -85,B 0,C 180,E1 -1099.335,E2 -1099.335} C_VEL
LIN {X 0,Y 594.361,Z 366.45,A -85,B 0,C 180,E1 -1101.504,E2 -1101.504} C_VEL
LIN {X 0,Y 594.382,Z 366.45,A -85,B 0,C 180,E1 -1104.446,E2 -1104.446} C_VEL
LIN {X 0,Y 594.384,Z 366.448,A -85,B 0,C 180,E1 -1106.7,E2 -1106.7} C_VEL
LIN {X 0,Y 594.379,Z 366.448,A -85,B 0,C 180,E1 -1108.999,E2 -1108.999} C_VEL
LIN {X 0,Y 594.373,Z 366.45,A -85,B 0,C 180,E1 -1111.643,E2 -1111.643} C_VEL
LIN {X 0,Y 594.388,Z 366.447,A -85,B 0,C 180,E1 -1114.58,E2 -1114.58} C_VEL
LIN {X 0,Y 594.385,Z 366.448,A -85,B 0,C 180,E1 -1117.609,E2 -1117.609} C_VEL
LIN {X 0,Y 594.368,Z 366.45,A -85,B 0,C 180,E1 -1120.567,E2 -1120.567} C_VEL
LIN {X 0,Y 594.362,Z 366.449,A -85,B 0,C 180,E1 -1123.3,E2 -1123.3} C_VEL
LIN {X 0,Y 594.364,Z 366.451,A -85,B 0,C 180,E1 -1126.161,E2 -1126.161} C_VEL
LIN {X 0,Y 594.382,Z 366.449,A -85,B 0,C 180,E1 -1128.537,E2 -1128.537} C_VEL
LIN {X 0,Y 594.376,Z 366.451,A -85,B 0,C 180,E1 -1131.297,E2 -1131.297} C_VEL
LIN {X 0,Y 594.453,Z 366.637,A -85,B 0,C 180,E1 -1133.973,E2 -1133.973} C_VEL
LIN {X 0,Y 594.596,Z 372.55,A -85,B 0,C 180,E1 -1135.831,E2 -1135.831} C_VEL
LIN {X 0,Y 594.593,Z 380.731,A -85,B 0,C 180,E1 -1138.324,E2 -1138.324} C_VEL
LIN {X 0,Y 594.504,Z 389.849,A -85,B 0,C 180,E1 -1141.022,E2 -1141.022} C_VEL
LIN {X 0,Y 594.495,Z 400.025,A -85,B 0,C 180,E1 -1143.956,E2 -1143.956} C_VEL
LIN {X 0,Y 594.414,Z 409.663,A -85,B 0,C 180,E1 -1146.667,E2 -1146.667} C_VEL
LIN {X 0,Y 594.404,Z 418.93,A -85,B 0,C 180,E1 -1149.225,E2 -1149.225} C_VEL
LIN {X 0,Y 594.36,Z 429.521,A -85,B 0,C 180,E1 -1152.095,E2 -1152.095} C_VEL
LIN {X 0,Y 594.305,Z 440.112,A -85,B 0,C 180,E1 -1154.92,E2 -1154.92} C_VEL
LIN {X 0,Y 594.267,Z 449.379,A -85,B 0,C 180,E1 -1157.362,E2 -1157.362} C_VEL
LIN {X 0,Y 594.31,Z 451.737,A -85,B 0,C 180,E1 -1157.943,E2 -1157.943} C_VEL
LIN {X 0,Y 594.69,Z 456.092,A -85,B 0,C 180,E1 -1158.021,E2 -1158.021} C_VEL
LIN {X 0,Y 594.625,Z 469.738,A -85,B 0,C 180,E1 -1158.344,E2 -1158.344} C_VEL
LIN {X 0,Y 594.553,Z 480.738,A -85,B 0,C 180,E1 -1158.724,E2 -1158.724} C_VEL
LIN {X 0,Y 594.495,Z 492.635,A -85,B 0,C 180,E1 -1159.269,E2 -1159.269} C_VEL
LIN {X 0,Y 594.476,Z 504.199,A -85,B 0,C 180,E1 -1159.958,E2 -1159.958} C_VEL
LIN {X 0,Y 594.414,Z 514.595,A -85,B 0,C 180,E1 -1160.73,E2 -1160.73} C_VEL
LIN {X 0,Y 594.383,Z 523.112,A -85,B 0,C 180,E1 -1161.501,E2 -1161.501} C_VEL
LIN {X 0,Y 594.347,Z 530.96,A -85,B 0,C 180,E1 -1162.355,E2 -1162.355} C_VEL
LIN {X 0,Y 594.283,Z 538.812,A -85,B 0,C 180,E1 -1163.408,E2 -1163.408} C_VEL
LIN {X 0,Y 594.289,Z 545.68,A -85,B 0,C 180,E1 -1164.571,E2 -1164.571} C_VEL
LIN {X 0,Y 594.27,Z 550.371,A -85,B 0,C 180,E1 -1165.591,E2 -1165.591} C_VEL
LIN {X 0,Y 594.267,Z 553.956,A -85,B 0,C 180,E1 -1166.61,E2 -1166.61} C_VEL
LIN {X 0,Y 594.226,Z 555.809,A -85,B 0,C 180,E1 -1167.288,E2 -1167.288} C_VEL
LIN {X 0,Y 594.242,Z 557.201,A -85,B 0,C 180,E1 -1167.967,E2 -1167.967} C_VEL
LIN {X 0,Y 594.239,Z 558.784,A -85,B 0,C 180,E1 -1169.322,E2 -1169.322} C_VEL
LIN {X 0,Y 594.236,Z 559,A -85,B 0,C 180,E1 -1170,E2 -1170} C_VEL
LIN {X 0,Y 594.247,Z 558.185,A -85,B 0,C 180,E1 -1171.355,E2 -1171.355} C_VEL
LIN {X 0,Y 594.242,Z 557.202,A -85,B 0,C 180,E1 -1172.033,E2 -1172.033} C_VEL
LIN {X 0,Y 594.226,Z 555.81,A -85,B 0,C 180,E1 -1172.711,E2 -1172.711} C_VEL
LIN {X 0,Y 594.289,Z 552.897,A -85,B 0,C 180,E1 -1173.729,E2 -1173.729} C_VEL
LIN {X 0,Y 594.241,Z 548.951,A -85,B 0,C 180,E1 -1174.749,E2 -1174.749} C_VEL
LIN {X 0,Y 594.304,Z 542.879,A -85,B 0,C 180,E1 -1175.939,E2 -1175.939} C_VEL
LIN {X 0,Y 594.308,Z 536.238,A -85,B 0,C 180,E1 -1176.962,E2 -1176.962} C_VEL
LIN {X 0,Y 594.359,Z 527.992,A -85,B 0,C 180,E1 -1177.986,E2 -1177.986} C_VEL
LIN {X 0,Y 594.382,Z 519.54,A -85,B 0,C 180,E1 -1178.842,E2 -1178.842} C_VEL
LIN {X 0,Y 594.434,Z 509.097,A -85,B 0,C 180,E1 -1179.699,E2 -1179.699} C_VEL
LIN {X 0,Y 594.463,Z 498.763,A -85,B 0,C 180,E1 -1180.386,E2 -1180.386} C_VEL
LIN {X 0,Y 594.505,Z 486.723,A -85,B 0,C 180,E1 -1181.021,E2 -1181.021} C_VEL
LIN {X 0,Y 594.564,Z 474.496,A -85,B 0,C 180,E1 -1181.505,E2 -1181.505} C_VEL
LIN {X 0,Y 594.68,Z 461.455,A -85,B 0,C 180,E1 -1181.871,E2 -1181.871} C_VEL
LIN {X 0,Y 594.446,Z 452.806,A -85,B 0,C 180,E1 -1182.039,E2 -1182.039} C_VEL
LIN {X 0,Y 594.294,Z 451.532,A -85,B 0,C 180,E1 -1182.073,E2 -1182.073} C_VEL
LIN {X 0,Y 594.31,Z 441.437,A -85,B 0,C 180,E1 -1184.729,E2 -1184.729} C_VEL
LIN {X 0,Y 594.335,Z 430.846,A -85,B 0,C 180,E1 -1187.549,E2 -1187.549} C_VEL
LIN {X 0,Y 594.384,Z 420.255,A -85,B 0,C 180,E1 -1190.414,E2 -1190.414} C_VEL
LIN {X 0,Y 594.404,Z 410.988,A -85,B 0,C 180,E1 -1192.965,E2 -1192.965} C_VEL
LIN {X 0,Y 594.475,Z 401.721,A -85,B 0,C 180,E1 -1195.563,E2 -1195.563} C_VEL
LIN {X 0,Y 594.494,Z 392.454,A -85,B 0,C 180,E1 -1198.22,E2 -1198.22} C_VEL
LIN {X 0,Y 594.528,Z 383.187,A -85,B 0,C 180,E1 -1200.944,E2 -1200.944} C_VEL
LIN {X 0,Y 594.637,Z 375.244,A -85,B 0,C 180,E1 -1203.337,E2 -1203.337} C_VEL
LIN {X 0,Y 594.583,Z 367.3,A -85,B 0,C 180,E1 -1205.808,E2 -1205.808} C_VEL
LIN {X 0,Y 594.405,Z 366.448,A -85,B 0,C 180,E1 -1206.135,E2 -1206.135} C_VEL
LIN {X 0,Y 594.374,Z 366.449,A -85,B 0,C 180,E1 -1208.805,E2 -1208.805} C_VEL
LIN {X 0,Y 594.379,Z 366.451,A -85,B 0,C 180,E1 -1211.848,E2 -1211.848} C_VEL
LIN {X 0,Y 594.377,Z 366.449,A -85,B 0,C 180,E1 -1214.235,E2 -1214.235} C_VEL
LIN {X 0,Y 594.356,Z 366.452,A -85,B 0,C 180,E1 -1217.147,E2 -1217.147} C_VEL
LIN {X 0,Y 594.367,Z 366.452,A -85,B 0,C 180,E1 -1219.433,E2 -1219.433} C_VEL
LIN {X 0,Y 594.386,Z 366.447,A -85,B 0,C 180,E1 -1222.39,E2 -1222.39} C_VEL
LIN {X 0,Y 594.38,Z 366.448,A -85,B 0,C 180,E1 -1224.671,E2 -1224.671} C_VEL
LIN {X 0,Y 594.372,Z 366.45,A -85,B 0,C 180,E1 -1227.087,E2 -1227.087} C_VEL
LIN {X 0,Y 594.379,Z 366.449,A -85,B 0,C 180,E1 -1229.671,E2 -1229.671} C_VEL
LIN {X 0,Y 594.383,Z 366.448,A -85,B 0,C 180,E1 -1232.539,E2 -1232.539} C_VEL
LIN {X 0,Y 594.369,Z 366.45,A -85,B 0,C 180,E1 -1234.807,E2 -1234.807} C_VEL
LIN {X 0,Y 594.357,Z 366.454,A -85,B 0,C 180,E1 -1237.264,E2 -1237.264} C_VEL
LIN {X 0,Y 594.373,Z 366.449,A -85,B 0,C 180,E1 -1239.946,E2 -1239.946} C_VEL
LIN {X 0,Y 594.386,Z 366.45,A -85,B 0,C 180,E1 -1242.807,E2 -1242.807} C_VEL
LIN {X 0,Y 594.38,Z 366.449,A -85,B 0,C 180,E1 -1245.825,E2 -1245.825} C_VEL
LIN {X 0,Y 594.387,Z 366.449,A -85,B 0,C 180,E1 -1248.404,E2 -1248.404} C_VEL
LIN {X 0,Y 594.397,Z 366.446,A -85,B 0,C 180,E1 -1251.158,E2 -1251.158} C_VEL
LIN {X 0,Y 594.398,Z 366.446,A -85,B 0,C 180,E1 -1253.299,E2 -1253.299} C_VEL
LIN {X 0,Y 594.359,Z 366.452,A -85,B 0,C 180,E1 -1255.932,E2 -1255.932} C_VEL
LIN {X 0,Y 594.378,Z 366.449,A -85,B 0,C 180,E1 -1258.645,E2 -1258.645} C_VEL
LIN {X 0,Y 594.377,Z 366.449,A -85,B 0,C 180,E1 -1261.355,E2 -1261.355} C_VEL
LIN {X 0,Y 594.38,Z 366.448,A -85,B 0,C 180,E1 -1263.389,E2 -1263.389} C_VEL
LIN {X 0,Y 594.368,Z 366.452,A -85,B 0,C 180,E1 -1266.109,E2 -1266.109} C_VEL
LIN {X 0,Y 594.398,Z 366.446,A -85,B 0,C 180,E1 -1268.842,E2 -1268.842} C_VEL
LIN {X 0,Y 594.387,Z 366.45,A -85,B 0,C 180,E1 -1271.596,E2 -1271.596} C_VEL
LIN {X 0,Y 594.38,Z 366.448,A -85,B 0,C 180,E1 -1274.377,E2 -1274.377} C_VEL
LIN {X 0,Y 594.354,Z 366.451,A -85,B 0,C 180,E1 -1275.333,E2 -1275.333} C_VEL
LIN {X 0,Y 593.686,Z 366.536,A -85,B 0,C 180,E1 -1275.899,E2 -1275.899} C_VEL
LIN {X 0,Y 590.832,Z 366.892,A -85,B 0,C 180,E1 -1276.817,E2 -1276.817} C_VEL
LIN {X 0,Y 588.426,Z 367.193,A -85,B 0,C 180,E1 -1277.556,E2 -1277.556} C_VEL
LIN {X 0,Y 587.399,Z 367.32,A -85,B 0,C 180,E1 -1278.126,E2 -1278.126} C_VEL
LIN {X 0,Y 587.319,Z 367.328,A -85,B 0,C 180,E1 -1278.319,E2 -1278.319} C_VEL
LIN {X 0,Y 587.349,Z 367.324,A -85,B 0,C 180,E1 -1281.045,E2 -1281.045} C_VEL
LIN {X 0,Y 587.332,Z 367.327,A -85,B 0,C 180,E1 -1284.007,E2 -1284.007} C_VEL
LIN {X 0,Y 587.356,Z 367.323,A -85,B 0,C 180,E1 -1286.278,E2 -1286.278} C_VEL
LIN {X 0,Y 587.345,Z 367.326,A -85,B 0,C 180,E1 -1289.135,E2 -1289.135} C_VEL
LIN {X 0,Y 587.349,Z 367.324,A -85,B 0,C 180,E1 -1291.838,E2 -1291.838} C_VEL
LIN {X 0,Y 587.354,Z 367.323,A -85,B 0,C 180,E1 -1294.35,E2 -1294.35} C_VEL
LIN {X 0,Y 587.349,Z 367.325,A -85,B 0,C 180,E1 -1296.747,E2 -1296.747} C_VEL
LIN {X 0,Y 587.341,Z 367.327,A -85,B 0,C 180,E1 -1299.36,E2 -1299.36} C_VEL
LIN {X 0,Y 587.33,Z 367.326,A -85,B 0,C 180,E1 -1302.109,E2 -1302.109} C_VEL
LIN {X 0,Y 587.312,Z 367.328,A -85,B 0,C 180,E1 -1305.09,E2 -1305.09} C_VEL
LIN {X 0,Y 587.35,Z 367.325,A -85,B 0,C 180,E1 -1307.929,E2 -1307.929} C_VEL
LIN {X 0,Y 587.33,Z 367.326,A -85,B 0,C 180,E1 -1311.059,E2 -1311.059} C_VEL
LIN {X 0,Y 587.351,Z 367.324,A -85,B 0,C 180,E1 -1313.293,E2 -1313.293} C_VEL
LIN {X 0,Y 587.361,Z 367.325,A -85,B 0,C 180,E1 -1315.781,E2 -1315.781} C_VEL
LIN {X 0,Y 587.35,Z 367.325,A -85,B 0,C 180,E1 -1318.233,E2 -1318.233} C_VEL
LIN {X 0,Y 587.351,Z 367.323,A -85,B 0,C 180,E1 -1320.867,E2 -1320.867} C_VEL
LIN {X 0,Y 587.364,Z 367.323,A -85,B 0,C 180,E1 -1323.819,E2 -1323.819} C_VEL
LIN {X 0,Y 587.34,Z 367.326,A -85,B 0,C 180,E1 -1325.994,E2 -1325.994} C_VEL
LIN {X 0,Y 587.321,Z 367.328,A -85,B 0,C 180,E1 -1328.226,E2 -1328.226} C_VEL
LIN {X 0,Y 587.351,Z 367.325,A -85,B 0,C 180,E1 -1331.152,E2 -1331.152} C_VEL
LIN {X 0,Y 587.324,Z 367.327,A -85,B 0,C 180,E1 -1334.025,E2 -1334.025} C_VEL
LIN {X 0,Y 587.366,Z 367.322,A -85,B 0,C 180,E1 -1336.155,E2 -1336.155} C_VEL
LIN {X 0,Y 587.342,Z 367.327,A -85,B 0,C 180,E1 -1338.963,E2 -1338.963} C_VEL
LIN {X 0,Y 587.37,Z 367.321,A -85,B 0,C 180,E1 -1341.745,E2 -1341.745} C_VEL
LIN {X 0,Y 587.362,Z 367.325,A -85,B 0,C 180,E1 -1344.507,E2 -1344.507} C_VEL
LIN {X 0,Y 587.241,Z 367.341,A -85,B 0,C 180,E1 -1347.256,E2 -1347.256} C_VEL
LIN {X 0,Y 587.28,Z 369.49,A -85,B 0,C 180,E1 -1349.315,E2 -1349.315} C_VEL
LIN {X 0,Y 587.222,Z 372.742,A -85,B 0,C 180,E1 -1352.058,E2 -1352.058} C_VEL
LIN {X 0,Y 587.198,Z 375.859,A -85,B 0,C 180,E1 -1354.806,E2 -1354.806} C_VEL
LIN {X 0,Y 587.182,Z 379.307,A -85,B 0,C 180,E1 -1357.566,E2 -1357.566} C_VEL
LIN {X 0,Y 587.143,Z 382.889,A -85,B 0,C 180,E1 -1360.343,E2 -1360.343} C_VEL
LIN {X 0,Y 587.16,Z 385.64,A -85,B 0,C 180,E1 -1362.442,E2 -1362.442} C_VEL
LIN {X 0,Y 587.144,Z 388.453,A -85,B 0,C 180,E1 -1364.558,E2 -1364.558} C_VEL
LIN {X 0,Y 587.126,Z 392.297,A -85,B 0,C 180,E1 -1367.413,E2 -1367.413} C_VEL
LIN {X 0,Y 587.139,Z 395.688,A -85,B 0,C 180,E1 -1369.901,E2 -1369.901} C_VEL
LIN {X 0,Y 587.721,Z 401.779,A -85,B 0,C 180,E1 -1370.04,E2 -1370.04} C_VEL
LIN {X 0,Y 587.625,Z 415.346,A -85,B 0,C 180,E1 -1370.431,E2 -1370.431} C_VEL
LIN {X 0,Y 587.523,Z 427.712,A -85,B 0,C 180,E1 -1370.938,E2 -1370.938} C_VEL
LIN {X 0,Y 587.493,Z 439.557,A -85,B 0,C 180,E1 -1371.583,E2 -1371.583} C_VEL
LIN {X 0,Y 587.407,Z 450.389,A -85,B 0,C 180,E1 -1372.325,E2 -1372.325} C_VEL
LIN {X 0,Y 587.333,Z 460.057,A -85,B 0,C 180,E1 -1373.145,E2 -1373.145} C_VEL
LIN {X 0,Y 587.298,Z 469.797,A -85,B 0,C 180,E1 -1374.172,E2 -1374.172} C_VEL
LIN {X 0,Y 587.239,Z 477.255,A -85,B 0,C 180,E1 -1375.141,E2 -1375.141} C_VEL
LIN {X 0,Y 587.209,Z 484.28,A -85,B 0,C 180,E1 -1376.284,E2 -1376.284} C_VEL
LIN {X 0,Y 587.19,Z 489.43,A -85,B 0,C 180,E1 -1377.355,E2 -1377.355} C_VEL
LIN {X 0,Y 587.159,Z 493.931,A -85,B 0,C 180,E1 -1378.605,E2 -1378.605} C_VEL
LIN {X 0,Y 587.138,Z 496.01,A -85,B 0,C 180,E1 -1379.391,E2 -1379.391} C_VEL
LIN {X 0,Y 587.155,Z 497.961,A -85,B 0,C 180,E1 -1380.479,E2 -1380.479} C_VEL
LIN {X 0,Y 587.131,Z 498.951,A -85,B 0,C 180,E1 -1381.801,E2 -1381.801} C_VEL
LIN {X 0,Y 587.138,Z 498.544,A -85,B 0,C 180,E1 -1383.081,E2 -1383.081} C_VEL
LIN {X 0,Y 587.136,Z 496.81,A -85,B 0,C 180,E1 -1384.317,E2 -1384.317} C_VEL
LIN {X 0,Y 587.161,Z 493.826,A -85,B 0,C 180,E1 -1385.518,E2 -1385.518} C_VEL
LIN {X 0,Y 587.195,Z 489.336,A -85,B 0,C 180,E1 -1386.757,E2 -1386.757} C_VEL
LIN {X 0,Y 587.188,Z 484.211,A -85,B 0,C 180,E1 -1387.819,E2 -1387.819} C_VEL
LIN {X 0,Y 587.226,Z 477.401,A -85,B 0,C 180,E1 -1388.928,E2 -1388.928} C_VEL
LIN {X 0,Y 587.276,Z 468.983,A -85,B 0,C 180,E1 -1390.013,E2 -1390.013} C_VEL
LIN {X 0,Y 587.354,Z 460.615,A -85,B 0,C 180,E1 -1390.891,E2 -1390.891} C_VEL
LIN {X 0,Y 587.417,Z 450.972,A -85,B 0,C 180,E1 -1391.721,E2 -1391.721} C_VEL
LIN {X 0,Y 587.439,Z 439.997,A -85,B 0,C 180,E1 -1392.481,E2 -1392.481} C_VEL
LIN {X 0,Y 587.478,Z 428.072,A -85,B 0,C 180,E1 -1393.135,E2 -1393.135} C_VEL
LIN {X 0,Y 587.601,Z 415.575,A -85,B 0,C 180,E1 -1393.652,E2 -1393.652} C_VEL
LIN {X 0,Y 587.689,Z 402,A -85,B 0,C 180,E1 -1394.046,E2 -1394.046} C_VEL
LIN {X 0,Y 587.391,Z 397.521,A -85,B 0,C 180,E1 -1394.148,E2 -1394.148} C_VEL
LIN {X 0,Y 587.116,Z 395.668,A -85,B 0,C 180,E1 -1394.204,E2 -1394.204} C_VEL
LIN {X 0,Y 587.124,Z 391.892,A -85,B 0,C 180,E1 -1396.976,E2 -1396.976} C_VEL
LIN {X 0,Y 587.12,Z 387.824,A -85,B 0,C 180,E1 -1400.004,E2 -1400.004} C_VEL
LIN {X 0,Y 587.126,Z 384.684,A -85,B 0,C 180,E1 -1402.376,E2 -1402.376} C_VEL
LIN {X 0,Y 587.124,Z 381.356,A -85,B 0,C 180,E1 -1404.93,E2 -1404.93} C_VEL
LIN {X 0,Y 587.158,Z 378.184,A -85,B 0,C 180,E1 -1407.409,E2 -1407.409} C_VEL
LIN {X 0,Y 587.193,Z 375.361,A -85,B 0,C 180,E1 -1409.822,E2 -1409.822} C_VEL
LIN {X 0,Y 587.21,Z 372.528,A -85,B 0,C 180,E1 -1412.332,E2 -1412.332} C_VEL
LIN {X 0,Y 587.239,Z 369.961,A -85,B 0,C 180,E1 -1414.479,E2 -1414.479} C_VEL
LIN {X 0,Y 587.245,Z 367.34,A -85,B 0,C 180,E1 -1416.738,E2 -1416.738} C_VEL
LIN {X 0,Y 587.343,Z 367.324,A -85,B 0,C 180,E1 -1418.963,E2 -1418.963} C_VEL
LIN {X 0,Y 587.324,Z 367.327,A -85,B 0,C 180,E1 -1421.873,E2 -1421.873} C_VEL
LIN {X 0,Y 587.317,Z 367.327,A -85,B 0,C 180,E1 -1424.024,E2 -1424.024} C_VEL
LIN {X 0,Y 587.353,Z 367.323,A -85,B 0,C 180,E1 -1426.154,E2 -1426.154} C_VEL
LIN {X 0,Y 587.341,Z 367.324,A -85,B 0,C 180,E1 -1428.962,E2 -1428.962} C_VEL
LIN {X 0,Y 587.365,Z 367.324,A -85,B 0,C 180,E1 -1431.745,E2 -1431.745} C_VEL
LIN {X 0,Y 587.355,Z 367.323,A -85,B 0,C 180,E1 -1434.507,E2 -1434.507} C_VEL
LIN {X 0,Y 587.371,Z 367.32,A -85,B 0,C 180,E1 -1437.257,E2 -1437.257} C_VEL
LIN {X 0,Y 587.372,Z 367.321,A -85,B 0,C 180,E1 -1440,E2 -1440} C_VEL
LIN {X 0,Y 587.37,Z 367.324,A -85,B 0,C 180,E1 -1442.743,E2 -1442.743} C_VEL
LIN {X 0,Y 587.354,Z 367.323,A -85,B 0,C 180,E1 -1445.493,E2 -1445.493} C_VEL
LIN {X 0,Y 587.361,Z 367.321,A -85,B 0,C 180,E1 -1448.255,E2 -1448.255} C_VEL
LIN {X 0,Y 587.356,Z 367.325,A -85,B 0,C 180,E1 -1451.141,E2 -1451.141} C_VEL
LIN {X 0,Y 587.357,Z 367.322,A -85,B 0,C 180,E1 -1454.261,E2 -1454.261} C_VEL
LIN {X 0,Y 587.354,Z 367.325,A -85,B 0,C 180,E1 -1457.406,E2 -1457.406} C_VEL
LIN {X 0,Y 587.325,Z 367.326,A -85,B 0,C 180,E1 -1460.305,E2 -1460.305} C_VEL
LIN {X 0,Y 587.316,Z 367.33,A -85,B 0,C 180,E1 -1463.259,E2 -1463.259} C_VEL
LIN {X 0,Y 587.334,Z 367.326,A -85,B 0,C 180,E1 -1465.517,E2 -1465.517} C_VEL
LIN {X 0,Y 587.344,Z 367.324,A -85,B 0,C 180,E1 -1467.818,E2 -1467.818} C_VEL
LIN {X 0,Y 587.329,Z 367.329,A -85,B 0,C 180,E1 -1470.51,E2 -1470.51} C_VEL
LIN {X 0,Y 587.323,Z 367.327,A -85,B 0,C 180,E1 -1473.398,E2 -1473.398} C_VEL
LIN {X 0,Y 587.288,Z 367.331,A -85,B 0,C 180,E1 -1475.9,E2 -1475.9} C_VEL
LIN {X 0,Y 587.332,Z 367.325,A -85,B 0,C 180,E1 -1478.479,E2 -1478.479} C_VEL
LIN {X 0,Y 587.333,Z 367.326,A -85,B 0,C 180,E1 -1481.157,E2 -1481.157} C_VEL
LIN {X 0,Y 587.323,Z 367.328,A -85,B 0,C 180,E1 -1484.114,E2 -1484.114} C_VEL
LIN {X 0,Y 587.312,Z 367.328,A -85,B 0,C 180,E1 -1486.994,E2 -1486.994} C_VEL
LIN {X 0,Y 587.316,Z 367.329,A -85,B 0,C 180,E1 -1489.747,E2 -1489.747} C_VEL
LIN {X 0,Y 587.339,Z 367.328,A -85,B 0,C 180,E1 -1492.393,E2 -1492.393} C_VEL
LIN {X 0,Y 587.381,Z 367.465,A -85,B 0,C 180,E1 -1493.736,E2 -1493.736} C_VEL
LIN {X 0,Y 587.67,Z 371.271,A -85,B 0,C 180,E1 -1494.968,E2 -1494.968} C_VEL
LIN {X 0,Y 587.589,Z 379.214,A -85,B 0,C 180,E1 -1497.437,E2 -1497.437} C_VEL
LIN {X 0,Y 587.554,Z 388.481,A -85,B 0,C 180,E1 -1500.238,E2 -1500.238} C_VEL
LIN {X 0,Y 587.418,Z 397.748,A -85,B 0,C 180,E1 -1502.959,E2 -1502.959} C_VEL
LIN {X 0,Y 587.443,Z 405.691,A -85,B 0,C 180,E1 -1505.246,E2 -1505.246} C_VEL
LIN {X 0,Y 587.388,Z 416.282,A -85,B 0,C 180,E1 -1508.229,E2 -1508.229} C_VEL
LIN {X 0,Y 587.311,Z 426.873,A -85,B 0,C 180,E1 -1511.15,E2 -1511.15} C_VEL
LIN {X 0,Y 587.262,Z 437.464,A -85,B 0,C 180,E1 -1514.023,E2 -1514.023} C_VEL
LIN {X 0,Y 587.233,Z 448.055,A -85,B 0,C 180,E1 -1516.857,E2 -1516.857} C_VEL
LIN {X 0,Y 587.217,Z 451.582,A -85,B 0,C 180,E1 -1517.792,E2 -1517.792} C_VEL
LIN {X 0,Y 587.746,Z 456.092,A -85,B 0,C 180,E1 -1517.877,E2 -1517.877} C_VEL
LIN {X 0,Y 587.672,Z 469.739,A -85,B 0,C 180,E1 -1518.204,E2 -1518.204} C_VEL
LIN {X 0,Y 587.569,Z 482.352,A -85,B 0,C 180,E1 -1518.654,E2 -1518.654} C_VEL
LIN {X 0,Y 587.494,Z 494.209,A -85,B 0,C 180,E1 -1519.227,E2 -1519.227} C_VEL
LIN {X 0,Y 587.468,Z 505.477,A -85,B 0,C 180,E1 -1519.924,E2 -1519.924} C_VEL
LIN {X 0,Y 587.384,Z 515.647,A -85,B 0,C 180,E1 -1520.705,E2 -1520.705} C_VEL
LIN {X 0,Y 587.34,Z 524.787,A -85,B 0,C 180,E1 -1521.571,E2 -1521.571} C_VEL
LIN {X 0,Y 587.259,Z 533.691,A -85,B 0,C 180,E1 -1522.608,E2 -1522.608} C_VEL
LIN {X 0,Y 587.195,Z 540.745,A -85,B 0,C 180,E1 -1523.627,E2 -1523.627} C_VEL
LIN {X 0,Y 587.211,Z 545.68,A -85,B 0,C 180,E1 -1524.506,E2 -1524.506} C_VEL
LIN {X 0,Y 587.188,Z 550.371,A -85,B 0,C 180,E1 -1525.538,E2 -1525.538} C_VEL
LIN {X 0,Y 587.193,Z 553.956,A -85,B 0,C 180,E1 -1526.569,E2 -1526.569} C_VEL
LIN {X 0,Y 587.132,Z 555.809,A -85,B 0,C 180,E1 -1527.256,E2 -1527.256} C_VEL
LIN {X 0,Y 587.141,Z 557.201,A -85,B 0,C 180,E1 -1527.942,E2 -1527.942} C_VEL
LIN {X 0,Y 587.14,Z 558.784,A -85,B 0,C 180,E1 -1529.314,E2 -1529.314} C_VEL
LIN {X 0,Y 587.137,Z 559,A -85,B 0,C 180,E1 -1530,E2 -1530} C_VEL
LIN {X 0,Y 587.147,Z 558.185,A -85,B 0,C 180,E1 -1531.372,E2 -1531.372} C_VEL
LIN {X 0,Y 587.141,Z 557.202,A -85,B 0,C 180,E1 -1532.058,E2 -1532.058} C_VEL
LIN {X 0,Y 587.132,Z 555.81,A -85,B 0,C 180,E1 -1532.744,E2 -1532.744} C_VEL
LIN {X 0,Y 587.213,Z 552.897,A -85,B 0,C 180,E1 -1533.774,E2 -1533.774} C_VEL
LIN {X 0,Y 587.147,Z 548.951,A -85,B 0,C 180,E1 -1534.806,E2 -1534.806} C_VEL
LIN {X 0,Y 587.217,Z 542.879,A -85,B 0,C 180,E1 -1536.011,E2 -1536.011} C_VEL
LIN {X 0,Y 587.244,Z 536.238,A -85,B 0,C 180,E1 -1537.046,E2 -1537.046} C_VEL
LIN {X 0,Y 587.299,Z 527.992,A -85,B 0,C 180,E1 -1538.083,E2 -1538.083} C_VEL
LIN {X 0,Y 587.343,Z 519.541,A -85,B 0,C 180,E1 -1538.949,E2 -1538.949} C_VEL
LIN {X 0,Y 587.421,Z 509.098,A -85,B 0,C 180,E1 -1539.816,E2 -1539.816} C_VEL
LIN {X 0,Y 587.478,Z 498.764,A -85,B 0,C 180,E1 -1540.511,E2 -1540.511} C_VEL
LIN {X 0,Y 587.531,Z 487.149,A -85,B 0,C 180,E1 -1541.134,E2 -1541.134} C_VEL
LIN {X 0,Y 587.624,Z 474.694,A -85,B 0,C 180,E1 -1541.636,E2 -1541.636} C_VEL
LIN {X 0,Y 587.717,Z 461.455,A -85,B 0,C 180,E1 -1542.013,E2 -1542.013} C_VEL
LIN {X 0,Y 587.548,Z 453.642,A -85,B 0,C 180,E1 -1542.17,E2 -1542.17} C_VEL
LIN {X 0,Y 587.204,Z 451.532,A -85,B 0,C 180,E1 -1542.221,E2 -1542.221} C_VEL
LIN {X 0,Y 587.257,Z 441.437,A -85,B 0,C 180,E1 -1544.91,E2 -1544.91} C_VEL
LIN {X 0,Y 587.302,Z 430.846,A -85,B 0,C 180,E1 -1547.766,E2 -1547.766} C_VEL
LIN {X 0,Y 587.376,Z 420.255,A -85,B 0,C 180,E1 -1550.668,E2 -1550.668} C_VEL
LIN {X 0,Y 587.388,Z 410.988,A -85,B 0,C 180,E1 -1553.255,E2 -1553.255} C_VEL
LIN {X 0,Y 587.485,Z 401.834,A -85,B 0,C 180,E1 -1555.857,E2 -1555.857} C_VEL
LIN {X 0,Y 587.467,Z 392.454,A -85,B 0,C 180,E1 -1558.589,E2 -1558.589} C_VEL
LIN {X 0,Y 587.565,Z 384.511,A -85,B 0,C 180,E1 -1560.952,E2 -1560.952} C_VEL
LIN {X 0,Y 587.687,Z 376.568,A -85,B 0,C 180,E1 -1563.373,E2 -1563.373} C_VEL
LIN {X 0,Y 587.622,Z 368.624,A -85,B 0,C 180,E1 -1565.876,E2 -1565.876} C_VEL
LIN {X 0,Y 587.374,Z 367.324,A -85,B 0,C 180,E1 -1566.317,E2 -1566.317} C_VEL
LIN {X 0,Y 587.328,Z 367.327,A -85,B 0,C 180,E1 -1569.36,E2 -1569.36} C_VEL
LIN {X 0,Y 587.33,Z 367.327,A -85,B 0,C 180,E1 -1572.107,E2 -1572.107} C_VEL
LIN {X 0,Y 587.311,Z 367.331,A -85,B 0,C 180,E1 -1575.088,E2 -1575.088} C_VEL
LIN {X 0,Y 587.347,Z 367.324,A -85,B 0,C 180,E1 -1577.927,E2 -1577.927} C_VEL
LIN {X 0,Y 587.329,Z 367.326,A -85,B 0,C 180,E1 -1581.057,E2 -1581.057} C_VEL
LIN {X 0,Y 587.349,Z 367.324,A -85,B 0,C 180,E1 -1583.291,E2 -1583.291} C_VEL
LIN {X 0,Y 587.364,Z 367.322,A -85,B 0,C 180,E1 -1585.78,E2 -1585.78} C_VEL
LIN {X 0,Y 587.347,Z 367.325,A -85,B 0,C 180,E1 -1588.231,E2 -1588.231} C_VEL
LIN {X 0,Y 587.347,Z 367.325,A -85,B 0,C 180,E1 -1590.865,E2 -1590.865} C_VEL
LIN {X 0,Y 587.352,Z 367.325,A -85,B 0,C 180,E1 -1593.818,E2 -1593.818} C_VEL
LIN {X 0,Y 587.331,Z 367.328,A -85,B 0,C 180,E1 -1595.993,E2 -1595.993} C_VEL
LIN {X 0,Y 587.339,Z 367.325,A -85,B 0,C 180,E1 -1598.963,E2 -1598.963} C_VEL
LIN {X 0,Y 587.324,Z 367.328,A -85,B 0,C 180,E1 -1601.873,E2 -1601.873} C_VEL
LIN {X 0,Y 587.323,Z 367.329,A -85,B 0,C 180,E1 -1604.025,E2 -1604.025} C_VEL
LIN {X 0,Y 587.352,Z 367.326,A -85,B 0,C 180,E1 -1606.154,E2 -1606.154} C_VEL
LIN {X 0,Y 587.34,Z 367.325,A -85,B 0,C 180,E1 -1608.962,E2 -1608.962} C_VEL
LIN {X 0,Y 587.362,Z 367.324,A -85,B 0,C 180,E1 -1611.745,E2 -1611.745} C_VEL
LIN {X 0,Y 587.35,Z 367.324,A -85,B 0,C 180,E1 -1614.507,E2 -1614.507} C_VEL
LIN {X 0,Y 587.367,Z 367.323,A -85,B 0,C 180,E1 -1617.257,E2 -1617.257} C_VEL
LIN {X 0,Y 587.37,Z 367.321,A -85,B 0,C 180,E1 -1620,E2 -1620} C_VEL
LIN {X 0,Y 587.373,Z 367.324,A -85,B 0,C 180,E1 -1622.743,E2 -1622.743} C_VEL
LIN {X 0,Y 587.352,Z 367.323,A -85,B 0,C 180,E1 -1625.493,E2 -1625.493} C_VEL
LIN {X 0,Y 587.363,Z 367.325,A -85,B 0,C 180,E1 -1628.255,E2 -1628.255} C_VEL
LIN {X 0,Y 587.353,Z 367.323,A -85,B 0,C 180,E1 -1631.142,E2 -1631.142} C_VEL
LIN {X 0,Y 587.355,Z 367.323,A -85,B 0,C 180,E1 -1634.261,E2 -1634.261} C_VEL
LIN {X 0,Y 587.35,Z 367.324,A -85,B 0,C 180,E1 -1637.406,E2 -1637.406} C_VEL
LIN {X 0,Y 587.319,Z 367.328,A -85,B 0,C 180,E1 -1638.319,E2 -1638.319} C_VEL
LIN {X 0,Y 586.667,Z 367.409,A -85,B 0,C 180,E1 -1638.891,E2 -1638.891} C_VEL
LIN {X 0,Y 583.837,Z 367.763,A -85,B 0,C 180,E1 -1639.82,E2 -1639.82} C_VEL
LIN {X 0,Y 581.428,Z 368.065,A -85,B 0,C 180,E1 -1640.567,E2 -1640.567} C_VEL
LIN {X 0,Y 580.375,Z 368.195,A -85,B 0,C 180,E1 -1641.143,E2 -1641.143} C_VEL
LIN {X 0,Y 580.28,Z 368.205,A -85,B 0,C 180,E1 -1641.338,E2 -1641.338} C_VEL
LIN {X 0,Y 580.294,Z 368.203,A -85,B 0,C 180,E1 -1644.317,E2 -1644.317} C_VEL
LIN {X 0,Y 580.304,Z 368.202,A -85,B 0,C 180,E1 -1646.622,E2 -1646.622} C_VEL
LIN {X 0,Y 580.297,Z 368.205,A -85,B 0,C 180,E1 -1649.311,E2 -1649.311} C_VEL
LIN {X 0,Y 580.296,Z 368.203,A -85,B 0,C 180,E1 -1652.201,E2 -1652.201} C_VEL
LIN {X 0,Y 580.298,Z 368.204,A -85,B 0,C 180,E1 -1654.696,E2 -1654.696} C_VEL
LIN {X 0,Y 580.296,Z 368.203,A -85,B 0,C 180,E1 -1657.269,E2 -1657.269} C_VEL
LIN {X 0,Y 580.294,Z 368.205,A -85,B 0,C 180,E1 -1660.272,E2 -1660.272} C_VEL
LIN {X 0,Y 580.272,Z 368.206,A -85,B 0,C 180,E1 -1662.707,E2 -1662.707} C_VEL
LIN {X 0,Y 580.271,Z 368.206,A -85,B 0,C 180,E1 -1665.609,E2 -1665.609} C_VEL
LIN {X 0,Y 580.312,Z 368.202,A -85,B 0,C 180,E1 -1668.235,E2 -1668.235} C_VEL
LIN {X 0,Y 580.286,Z 368.203,A -85,B 0,C 180,E1 -1670.967,E2 -1670.967} C_VEL
LIN {X 0,Y 580.28,Z 368.207,A -85,B 0,C 180,E1 -1673.598,E2 -1673.598} C_VEL
LIN {X 0,Y 580.316,Z 368.2,A -85,B 0,C 180,E1 -1676.146,E2 -1676.146} C_VEL
LIN {X 0,Y 580.287,Z 368.203,A -85,B 0,C 180,E1 -1678.616,E2 -1678.616} C_VEL
LIN {X 0,Y 580.294,Z 368.203,A -85,B 0,C 180,E1 -1681.025,E2 -1681.025} C_VEL
LIN {X 0,Y 580.294,Z 368.205,A -85,B 0,C 180,E1 -1683.666,E2 -1683.666} C_VEL
LIN {X 0,Y 580.304,Z 368.203,A -85,B 0,C 180,E1 -1685.685,E2 -1685.685} C_VEL
LIN {X 0,Y 580.273,Z 368.208,A -85,B 0,C 180,E1 -1687.948,E2 -1687.948} C_VEL
LIN {X 0,Y 580.3,Z 368.202,A -85,B 0,C 180,E1 -1690.914,E2 -1690.914} C_VEL
LIN {X 0,Y 580.275,Z 368.206,A -85,B 0,C 180,E1 -1693.826,E2 -1693.826} C_VEL
LIN {X 0,Y 580.331,Z 368.199,A -85,B 0,C 180,E1 -1695.984,E2 -1695.984} C_VEL
LIN {X 0,Y 580.309,Z 368.202,A -85,B 0,C 180,E1 -1698.827,E2 -1698.827} C_VEL
LIN {X 0,Y 580.333,Z 368.198,A -85,B 0,C 180,E1 -1701.644,E2 -1701.644} C_VEL
LIN {X 0,Y 580.328,Z 368.2,A -85,B 0,C 180,E1 -1704.441,E2 -1704.441} C_VEL
LIN {X 0,Y 580.198,Z 368.218,A -85,B 0,C 180,E1 -1707.223,E2 -1707.223} C_VEL
LIN {X 0,Y 580.183,Z 368.477,A -85,B 0,C 180,E1 -1707.918,E2 -1707.918} C_VEL
LIN {X 0,Y 580.224,Z 370.892,A -85,B 0,C 180,E1 -1710,E2 -1710} C_VEL
LIN {X 0,Y 580.143,Z 373.375,A -85,B 0,C 180,E1 -1712.083,E2 -1712.083} C_VEL
LIN {X 0,Y 580.144,Z 376.501,A -85,B 0,C 180,E1 -1714.865,E2 -1714.865} C_VEL
LIN {X 0,Y 580.097,Z 379.825,A -85,B 0,C 180,E1 -1717.658,E2 -1717.658} C_VEL
LIN {X 0,Y 580.062,Z 383.412,A -85,B 0,C 180,E1 -1720.471,E2 -1720.471} C_VEL
LIN {X 0,Y 580.071,Z 386.167,A -85,B 0,C 180,E1 -1722.596,E2 -1722.596} C_VEL
LIN {X 0,Y 580.053,Z 388.984,A -85,B 0,C 180,E1 -1724.74,E2 -1724.74} C_VEL
LIN {X 0,Y 580.04,Z 391.863,A -85,B 0,C 180,E1 -1726.905,E2 -1726.905} C_VEL
LIN {X 0,Y 580.051,Z 395.673,A -85,B 0,C 180,E1 -1729.739,E2 -1729.739} C_VEL
LIN {X 0,Y 580.771,Z 401.939,A -85,B 0,C 180,E1 -1729.898,E2 -1729.898} C_VEL
LIN {X 0,Y 580.663,Z 414.79,A -85,B 0,C 180,E1 -1730.271,E2 -1730.271} C_VEL
LIN {X 0,Y 580.607,Z 426.007,A -85,B 0,C 180,E1 -1730.724,E2 -1730.724} C_VEL
LIN {X 0,Y 580.542,Z 436.939,A -85,B 0,C 180,E1 -1731.295,E2 -1731.295} C_VEL
LIN {X 0,Y 580.427,Z 448.26,A -85,B 0,C 180,E1 -1732.046,E2 -1732.046} C_VEL
LIN {X 0,Y 580.307,Z 458.988,A -85,B 0,C 180,E1 -1732.937,E2 -1732.937} C_VEL
LIN {X 0,Y 580.241,Z 466.979,A -85,B 0,C 180,E1 -1733.749,E2 -1733.749} C_VEL
LIN {X 0,Y 580.203,Z 474.758,A -85,B 0,C 180,E1 -1734.704,E2 -1734.704} C_VEL
LIN {X 0,Y 580.137,Z 482.275,A -85,B 0,C 180,E1 -1735.856,E2 -1735.856} C_VEL
LIN {X 0,Y 580.1,Z 488.24,A -85,B 0,C 180,E1 -1737.021,E2 -1737.021} C_VEL
LIN {X 0,Y 580.06,Z 492.811,A -85,B 0,C 180,E1 -1738.198,E2 -1738.198} C_VEL
LIN {X 0,Y 580.073,Z 495.813,A -85,B 0,C 180,E1 -1739.269,E2 -1739.269} C_VEL
LIN {X 0,Y 580.064,Z 498.186,A -85,B 0,C 180,E1 -1740.657,E2 -1740.657} C_VEL
LIN {X 0,Y 580.043,Z 498.994,A -85,B 0,C 180,E1 -1741.989,E2 -1741.989} C_VEL
LIN {X 0,Y 580.058,Z 498.359,A -85,B 0,C 180,E1 -1743.279,E2 -1743.279} C_VEL
LIN {X 0,Y 580.051,Z 496.444,A -85,B 0,C 180,E1 -1744.522,E2 -1744.522} C_VEL
LIN {X 0,Y 580.063,Z 493.31,A -85,B 0,C 180,E1 -1745.731,E2 -1745.731} C_VEL
LIN {X 0,Y 580.095,Z 488.962,A -85,B 0,C 180,E1 -1746.907,E2 -1746.907} C_VEL
LIN {X 0,Y 580.144,Z 482.721,A -85,B 0,C 180,E1 -1748.157,E2 -1748.157} C_VEL
LIN {X 0,Y 580.19,Z 475.205,A -85,B 0,C 180,E1 -1749.323,E2 -1749.323} C_VEL
LIN {X 0,Y 580.247,Z 466.841,A -85,B 0,C 180,E1 -1750.356,E2 -1750.356} C_VEL
LIN {X 0,Y 580.349,Z 456.938,A -85,B 0,C 180,E1 -1751.338,E2 -1751.338} C_VEL
LIN {X 0,Y 580.401,Z 447.472,A -85,B 0,C 180,E1 -1752.103,E2 -1752.103} C_VEL
LIN {X 0,Y 580.433,Z 436.717,A -85,B 0,C 180,E1 -1752.809,E2 -1752.809} C_VEL
LIN {X 0,Y 580.565,Z 424.808,A -85,B 0,C 180,E1 -1753.42,E2 -1753.42} C_VEL
LIN {X 0,Y 580.701,Z 412.46,A -85,B 0,C 180,E1 -1753.898,E2 -1753.898} C_VEL
LIN {X 0,Y 580.673,Z 399.807,A -85,B 0,C 180,E1 -1754.245,E2 -1754.245} C_VEL
LIN {X 0,Y 580.019,Z 395.676,A -85,B 0,C 180,E1 -1754.35,E2 -1754.35} C_VEL
LIN {X 0,Y 580.02,Z 391.75,A -85,B 0,C 180,E1 -1757.27,E2 -1757.27} C_VEL
LIN {X 0,Y 580.028,Z 388.069,A -85,B 0,C 180,E1 -1760.045,E2 -1760.045} C_VEL
LIN {X 0,Y 580.038,Z 384.084,A -85,B 0,C 180,E1 -1763.099,E2 -1763.099} C_VEL
LIN {X 0,Y 580.05,Z 381.038,A -85,B 0,C 180,E1 -1765.476,E2 -1765.476} C_VEL
LIN {X 0,Y 580.102,Z 377.995,A -85,B 0,C 180,E1 -1768,E2 -1768} C_VEL
LIN {X 0,Y 580.147,Z 375.044,A -85,B 0,C 180,E1 -1770.716,E2 -1770.716} C_VEL
LIN {X 0,Y 580.173,Z 371.506,A -85,B 0,C 180,E1 -1773.688,E2 -1773.688} C_VEL
LIN {X 0,Y 580.164,Z 368.339,A -85,B 0,C 180,E1 -1776.437,E2 -1776.437} C_VEL
LIN {X 0,Y 580.311,Z 368.201,A -85,B 0,C 180,E1 -1778.83,E2 -1778.83} C_VEL
LIN {X 0,Y 580.276,Z 368.204,A -85,B 0,C 180,E1 -1781.645,E2 -1781.645} C_VEL
LIN {X 0,Y 580.272,Z 368.205,A -85,B 0,C 180,E1 -1783.825,E2 -1783.825} C_VEL
LIN {X 0,Y 580.319,Z 368.201,A -85,B 0,C 180,E1 -1785.983,E2 -1785.983} C_VEL
LIN {X 0,Y 580.326,Z 368.198,A -85,B 0,C 180,E1 -1788.827,E2 -1788.827} C_VEL
LIN {X 0,Y 580.329,Z 368.199,A -85,B 0,C 180,E1 -1791.644,E2 -1791.644} C_VEL
LIN {X 0,Y 580.32,Z 368.2,A -85,B 0,C 180,E1 -1794.44,E2 -1794.44} C_VEL
LIN {X 0,Y 580.337,Z 368.196,A -85,B 0,C 180,E1 -1797.223,E2 -1797.223} C_VEL
LIN {X 0,Y 580.341,Z 368.196,A -85,B 0,C 180,E1 -1800,E2 -1800} C_VEL
LIN {X 0,Y 580.336,Z 368.2,A -85,B 0,C 180,E1 -1802.776,E2 -1802.776} C_VEL
LIN {X 0,Y 580.319,Z 368.199,A -85,B 0,C 180,E1 -1805.56,E2 -1805.56} C_VEL
LIN {X 0,Y 580.325,Z 368.198,A -85,B 0,C 180,E1 -1808.356,E2 -1808.356} C_VEL
LIN {X 0,Y 580.327,Z 368.201,A -85,B 0,C 180,E1 -1811.208,E2 -1811.208} C_VEL
LIN {X 0,Y 580.308,Z 368.2,A -85,B 0,C 180,E1 -1814.339,E2 -1814.339} C_VEL
LIN {X 0,Y 580.308,Z 368.2,A -85,B 0,C 180,E1 -1816.915,E2 -1816.915} C_VEL
LIN {X 0,Y 580.3,Z 368.204,A -85,B 0,C 180,E1 -1819.823,E2 -1819.823} C_VEL
LIN {X 0,Y 580.291,Z 368.202,A -85,B 0,C 180,E1 -1822.803,E2 -1822.803} C_VEL
LIN {X 0,Y 580.303,Z 368.201,A -85,B 0,C 180,E1 -1825.08,E2 -1825.08} C_VEL
LIN {X 0,Y 580.315,Z 368.2,A -85,B 0,C 180,E1 -1827.864,E2 -1827.864} C_VEL
LIN {X 0,Y 580.277,Z 368.207,A -85,B 0,C 180,E1 -1830.695,E2 -1830.695} C_VEL
LIN {X 0,Y 580.279,Z 368.205,A -85,B 0,C 180,E1 -1833.314,E2 -1833.314} C_VEL
LIN {X 0,Y 580.244,Z 368.21,A -85,B 0,C 180,E1 -1835.757,E2 -1835.757} C_VEL
LIN {X 0,Y 580.286,Z 368.204,A -85,B 0,C 180,E1 -1838.147,E2 -1838.147} C_VEL
LIN {X 0,Y 580.297,Z 368.202,A -85,B 0,C 180,E1 -1840.844,E2 -1840.844} C_VEL
LIN {X 0,Y 580.276,Z 368.205,A -85,B 0,C 180,E1 -1843.658,E2 -1843.658} C_VEL
LIN {X 0,Y 580.274,Z 368.206,A -85,B 0,C 180,E1 -1846.61,E2 -1846.61} C_VEL
LIN {X 0,Y 580.298,Z 368.203,A -85,B 0,C 180,E1 -1849.157,E2 -1849.157} C_VEL
LIN {X 0,Y 580.285,Z 368.204,A -85,B 0,C 180,E1 -1851.928,E2 -1851.928} C_VEL
LIN {X 0,Y 580.347,Z 368.33,A -85,B 0,C 180,E1 -1853.507,E2 -1853.507} C_VEL
LIN {X 0,Y 580.72,Z 371.271,A -85,B 0,C 180,E1 -1854.486,E2 -1854.486} C_VEL
LIN {X 0,Y 580.673,Z 379.214,A -85,B 0,C 180,E1 -1857,E2 -1857} C_VEL
LIN {X 0,Y 580.552,Z 387.157,A -85,B 0,C 180,E1 -1859.44,E2 -1859.44} C_VEL
LIN {X 0,Y 580.506,Z 396.034,A -85,B 0,C 180,E1 -1862.103,E2 -1862.103} C_VEL
LIN {X 0,Y 580.419,Z 405.691,A -85,B 0,C 180,E1 -1864.926,E2 -1864.926} C_VEL
LIN {X 0,Y 580.37,Z 416.282,A -85,B 0,C 180,E1 -1867.952,E2 -1867.952} C_VEL
LIN {X 0,Y 580.266,Z 426.873,A -85,B 0,C 180,E1 -1870.912,E2 -1870.912} C_VEL
LIN {X 0,Y 580.221,Z 437.464,A -85,B 0,C 180,E1 -1873.824,E2 -1873.824} C_VEL
LIN {X 0,Y 580.183,Z 448.055,A -85,B 0,C 180,E1 -1876.694,E2 -1876.694} C_VEL
LIN {X 0,Y 580.128,Z 451.53,A -85,B 0,C 180,E1 -1877.627,E2 -1877.627} C_VEL
LIN {X 0,Y 580.806,Z 457.234,A -85,B 0,C 180,E1 -1877.753,E2 -1877.753} C_VEL
LIN {X 0,Y 580.735,Z 470.499,A -85,B 0,C 180,E1 -1878.083,E2 -1878.083} C_VEL
LIN {X 0,Y 580.602,Z 482.579,A -85,B 0,C 180,E1 -1878.526,E2 -1878.526} C_VEL
LIN {X 0,Y 580.497,Z 494.21,A -85,B 0,C 180,E1 -1879.096,E2 -1879.096} C_VEL
LIN {X 0,Y 580.458,Z 505.477,A -85,B 0,C 180,E1 -1879.801,E2 -1879.801} C_VEL
LIN {X 0,Y 580.352,Z 515.647,A -85,B 0,C 180,E1 -1880.591,E2 -1880.591} C_VEL
LIN {X 0,Y 580.279,Z 524.787,A -85,B 0,C 180,E1 -1881.468,E2 -1881.468} C_VEL
LIN {X 0,Y 580.199,Z 533.691,A -85,B 0,C 180,E1 -1882.518,E2 -1882.518} C_VEL
LIN {X 0,Y 580.12,Z 540.466,A -85,B 0,C 180,E1 -1883.505,E2 -1883.505} C_VEL
LIN {X 0,Y 580.139,Z 545.68,A -85,B 0,C 180,E1 -1884.438,E2 -1884.438} C_VEL
LIN {X 0,Y 580.108,Z 550.371,A -85,B 0,C 180,E1 -1885.483,E2 -1885.483} C_VEL
LIN {X 0,Y 580.123,Z 553.956,A -85,B 0,C 180,E1 -1886.527,E2 -1886.527} C_VEL
LIN {X 0,Y 580.043,Z 555.808,A -85,B 0,C 180,E1 -1887.222,E2 -1887.222} C_VEL
LIN {X 0,Y 580.04,Z 557.201,A -85,B 0,C 180,E1 -1887.917,E2 -1887.917} C_VEL
LIN {X 0,Y 580.04,Z 558.784,A -85,B 0,C 180,E1 -1889.306,E2 -1889.306} C_VEL
LIN {X 0,Y 580.037,Z 559,A -85,B 0,C 180,E1 -1890,E2 -1890} C_VEL
LIN {X 0,Y 580.047,Z 558.185,A -85,B 0,C 180,E1 -1891.388,E2 -1891.388} C_VEL
LIN {X 0,Y 580.04,Z 557.202,A -85,B 0,C 180,E1 -1892.083,E2 -1892.083} C_VEL
LIN {X 0,Y 580.043,Z 555.81,A -85,B 0,C 180,E1 -1892.778,E2 -1892.778} C_VEL
LIN {X 0,Y 580.11,Z 552.897,A -85,B 0,C 180,E1 -1893.82,E2 -1893.82} C_VEL
LIN {X 0,Y 580.053,Z 548.951,A -85,B 0,C 180,E1 -1894.865,E2 -1894.865} C_VEL
LIN {X 0,Y 580.139,Z 542.879,A -85,B 0,C 180,E1 -1896.085,E2 -1896.085} C_VEL
LIN {X 0,Y 580.184,Z 536.238,A -85,B 0,C 180,E1 -1897.132,E2 -1897.132} C_VEL
LIN {X 0,Y 580.25,Z 527.992,A -85,B 0,C 180,E1 -1898.182,E2 -1898.182} C_VEL
LIN {X 0,Y 580.308,Z 519.541,A -85,B 0,C 180,E1 -1899.058,E2 -1899.058} C_VEL
LIN {X 0,Y 580.423,Z 509.098,A -85,B 0,C 180,E1 -1899.935,E2 -1899.935} C_VEL
LIN {X 0,Y 580.499,Z 498.765,A -85,B 0,C 180,E1 -1900.639,E2 -1900.639} C_VEL
LIN {X 0,Y 580.562,Z 487.602,A -85,B 0,C 180,E1 -1901.247,E2 -1901.247} C_VEL
LIN {X 0,Y 580.662,Z 475.779,A -85,B 0,C 180,E1 -1901.74,E2 -1901.74} C_VEL
LIN {X 0,Y 580.775,Z 462.369,A -85,B 0,C 180,E1 -1902.137,E2 -1902.137} C_VEL
LIN {X 0,Y 580.602,Z 454.357,A -85,B 0,C 180,E1 -1902.307,E2 -1902.307} C_VEL
LIN {X 0,Y 580.128,Z 451.532,A -85,B 0,C 180,E1 -1902.373,E2 -1902.373} C_VEL
LIN {X 0,Y 580.217,Z 441.437,A -85,B 0,C 180,E1 -1905.095,E2 -1905.095} C_VEL
LIN {X 0,Y 580.254,Z 430.846,A -85,B 0,C 180,E1 -1907.99,E2 -1907.99} C_VEL
LIN {X 0,Y 580.332,Z 420.494,A -85,B 0,C 180,E1 -1910.864,E2 -1910.864} C_VEL
LIN {X 0,Y 580.383,Z 410.988,A -85,B 0,C 180,E1 -1913.553,E2 -1913.553} C_VEL
LIN {X 0,Y 580.479,Z 401.224,A -85,B 0,C 180,E1 -1916.371,E2 -1916.371} C_VEL
LIN {X 0,Y 580.532,Z 391.162,A -85,B 0,C 180,E1 -1919.35,E2 -1919.35} C_VEL
LIN {X 0,Y 580.666,Z 381.863,A -85,B 0,C 180,E1 -1922.177,E2 -1922.177} C_VEL
LIN {X 0,Y 580.71,Z 373.92,A -85,B 0,C 180,E1 -1924.667,E2 -1924.667} C_VEL
LIN {X 0,Y 580.691,Z 370.337,A -85,B 0,C 180,E1 -1925.817,E2 -1925.817} C_VEL
LIN {X 0,Y 580.32,Z 368.2,A -85,B 0,C 180,E1 -1926.59,E2 -1926.59} C_VEL
LIN {X 0,Y 580.293,Z 368.203,A -85,B 0,C 180,E1 -1929.185,E2 -1929.185} C_VEL
LIN {X 0,Y 580.31,Z 368.203,A -85,B 0,C 180,E1 -1931.765,E2 -1931.765} C_VEL
LIN {X 0,Y 580.264,Z 368.206,A -85,B 0,C 180,E1 -1934.625,E2 -1934.625} C_VEL
LIN {X 0,Y 580.28,Z 368.205,A -85,B 0,C 180,E1 -1937.627,E2 -1937.627} C_VEL
LIN {X 0,Y 580.288,Z 368.203,A -85,B 0,C 180,E1 -1940.067,E2 -1940.067} C_VEL
LIN {X 0,Y 580.297,Z 368.204,A -85,B 0,C 180,E1 -1943.064,E2 -1943.064} C_VEL
LIN {X 0,Y 580.3,Z 368.202,A -85,B 0,C 180,E1 -1945.439,E2 -1945.439} C_VEL
LIN {X 0,Y 580.302,Z 368.201,A -85,B 0,C 180,E1 -1947.967,E2 -1947.967} C_VEL
LIN {X 0,Y 580.298,Z 368.205,A -85,B 0,C 180,E1 -1950.689,E2 -1950.689} C_VEL
LIN {X 0,Y 580.32,Z 368.2,A -85,B 0,C 180,E1 -1953.658,E2 -1953.658} C_VEL
LIN {X 0,Y 580.273,Z 368.206,A -85,B 0,C 180,E1 -1956.442,E2 -1956.442} C_VEL
LIN {X 0,Y 580.277,Z 368.207,A -85,B 0,C 180,E1 -1959.437,E2 -1959.437} C_VEL
LIN {X 0,Y 580.277,Z 368.207,A -85,B 0,C 180,E1 -1961.645,E2 -1961.645} C_VEL
LIN {X 0,Y 580.276,Z 368.207,A -85,B 0,C 180,E1 -1963.825,E2 -1963.825} C_VEL
LIN {X 0,Y 580.318,Z 368.201,A -85,B 0,C 180,E1 -1965.983,E2 -1965.983} C_VEL
LIN {X 0,Y 580.322,Z 368.199,A -85,B 0,C 180,E1 -1968.827,E2 -1968.827} C_VEL
LIN {X 0,Y 580.326,Z 368.201,A -85,B 0,C 180,E1 -1971.644,E2 -1971.644} C_VEL
LIN {X 0,Y 580.316,Z 368.2,A -85,B 0,C 180,E1 -1974.44,E2 -1974.44} C_VEL
LIN {X 0,Y 580.333,Z 368.2,A -85,B 0,C 180,E1 -1977.224,E2 -1977.224} C_VEL
LIN {X 0,Y 580.34,Z 368.197,A -85,B 0,C 180,E1 -1980,E2 -1980} C_VEL
LIN {X 0,Y 580.338,Z 368.199,A -85,B 0,C 180,E1 -1982.777,E2 -1982.777} C_VEL
LIN {X 0,Y 580.318,Z 368.199,A -85,B 0,C 180,E1 -1985.56,E2 -1985.56} C_VEL
LIN {X 0,Y 580.328,Z 368.2,A -85,B 0,C 180,E1 -1988.356,E2 -1988.356} C_VEL
LIN {X 0,Y 580.324,Z 368.199,A -85,B 0,C 180,E1 -1991.209,E2 -1991.209} C_VEL
LIN {X 0,Y 580.306,Z 368.201,A -85,B 0,C 180,E1 -1994.339,E2 -1994.339} C_VEL
LIN {X 0,Y 580.305,Z 368.203,A -85,B 0,C 180,E1 -1996.915,E2 -1996.915} C_VEL
LIN {X 0,Y 580.301,Z 368.202,A -85,B 0,C 180,E1 -1999.823,E2 -1999.823} C_VEL
LIN {X 0,Y 580.28,Z 368.205,A -85,B 0,C 180,E1 -2001.338,E2 -2001.338} C_VEL
LIN {X 0,Y 579.582,Z 368.292,A -85,B 0,C 180,E1 -2001.917,E2 -2001.917} C_VEL
LIN {X 0,Y 576.705,Z 368.65,A -85,B 0,C 180,E1 -2002.857,E2 -2002.857} C_VEL
LIN {X 0,Y 574.309,Z 368.95,A -85,B 0,C 180,E1 -2003.613,E2 -2003.613} C_VEL
LIN {X 0,Y 573.31,Z 369.073,A -85,B 0,C 180,E1 -2004.197,E2 -2004.197} C_VEL
LIN {X 0,Y 573.243,Z 369.081,A -85,B 0,C 180,E1 -2004.395,E2 -2004.395} C_VEL
LIN {X 0,Y 573.261,Z 369.081,A -85,B 0,C 180,E1 -2006.976,E2 -2006.976} C_VEL
LIN {X 0,Y 573.242,Z 369.082,A -85,B 0,C 180,E1 -2009.489,E2 -2009.489} C_VEL
LIN {X 0,Y 573.249,Z 369.081,A -85,B 0,C 180,E1 -2012.23,E2 -2012.23} C_VEL
LIN {X 0,Y 573.248,Z 369.083,A -85,B 0,C 180,E1 -2014.775,E2 -2014.775} C_VEL
LIN {X 0,Y 573.25,Z 369.081,A -85,B 0,C 180,E1 -2017.167,E2 -2017.167} C_VEL
LIN {X 0,Y 573.243,Z 369.081,A -85,B 0,C 180,E1 -2019.608,E2 -2019.608} C_VEL
LIN {X 0,Y 573.235,Z 369.083,A -85,B 0,C 180,E1 -2022.642,E2 -2022.642} C_VEL
LIN {X 0,Y 573.236,Z 369.083,A -85,B 0,C 180,E1 -2025.668,E2 -2025.668} C_VEL
LIN {X 0,Y 573.242,Z 369.081,A -85,B 0,C 180,E1 -2028.545,E2 -2028.545} C_VEL
LIN {X 0,Y 573.245,Z 369.082,A -85,B 0,C 180,E1 -2031.3,E2 -2031.3} C_VEL
LIN {X 0,Y 573.244,Z 369.081,A -85,B 0,C 180,E1 -2034.015,E2 -2034.015} C_VEL
LIN {X 0,Y 573.285,Z 369.076,A -85,B 0,C 180,E1 -2036.52,E2 -2036.52} C_VEL
LIN {X 0,Y 573.239,Z 369.084,A -85,B 0,C 180,E1 -2039.117,E2 -2039.117} C_VEL
LIN {X 0,Y 573.248,Z 369.08,A -85,B 0,C 180,E1 -2041.973,E2 -2041.973} C_VEL
LIN {X 0,Y 573.258,Z 369.081,A -85,B 0,C 180,E1 -2044.591,E2 -2044.591} C_VEL
LIN {X 0,Y 573.238,Z 369.082,A -85,B 0,C 180,E1 -2047.663,E2 -2047.663} C_VEL
LIN {X 0,Y 573.268,Z 369.077,A -85,B 0,C 180,E1 -2050.671,E2 -2050.671} C_VEL
LIN {X 0,Y 573.248,Z 369.083,A -85,B 0,C 180,E1 -2053.622,E2 -2053.622} C_VEL
LIN {X 0,Y 573.278,Z 369.079,A -85,B 0,C 180,E1 -2055.808,E2 -2055.808} C_VEL
LIN {X 0,Y 573.267,Z 369.078,A -85,B 0,C 180,E1 -2058.746,E2 -2058.746} C_VEL
LIN {X 0,Y 573.288,Z 369.076,A -85,B 0,C 180,E1 -2061.541,E2 -2061.541} C_VEL
LIN {X 0,Y 573.296,Z 369.076,A -85,B 0,C 180,E1 -2064.372,E2 -2064.372} C_VEL
LIN {X 0,Y 573.154,Z 369.095,A -85,B 0,C 180,E1 -2067.189,E2 -2067.189} C_VEL
LIN {X 0,Y 573.111,Z 369.102,A -85,B 0,C 180,E1 -2067.892,E2 -2067.892} C_VEL
LIN {X 0,Y 573.175,Z 371.52,A -85,B 0,C 180,E1 -2070,E2 -2070} C_VEL
LIN {X 0,Y 573.061,Z 373.968,A -85,B 0,C 180,E1 -2072.109,E2 -2072.109} C_VEL
LIN {X 0,Y 573.071,Z 377.143,A -85,B 0,C 180,E1 -2074.925,E2 -2074.925} C_VEL
LIN {X 0,Y 573.031,Z 380.392,A -85,B 0,C 180,E1 -2077.753,E2 -2077.753} C_VEL
LIN {X 0,Y 572.992,Z 383.934,A -85,B 0,C 180,E1 -2080.602,E2 -2080.602} C_VEL
LIN {X 0,Y 572.989,Z 387.627,A -85,B 0,C 180,E1 -2083.476,E2 -2083.476} C_VEL
LIN {X 0,Y 572.966,Z 391.431,A -85,B 0,C 180,E1 -2086.386,E2 -2086.386} C_VEL
LIN {X 0,Y 572.962,Z 395.596,A -85,B 0,C 180,E1 -2089.527,E2 -2089.527} C_VEL
LIN {X 0,Y 572.959,Z 395.69,A -85,B 0,C 180,E1 -2089.597,E2 -2089.597} C_VEL
LIN {X 0,Y 573.831,Z 402.086,A -85,B 0,C 180,E1 -2089.752,E2 -2089.752} C_VEL
LIN {X 0,Y 573.706,Z 415.582,A -85,B 0,C 180,E1 -2090.153,E2 -2090.153} C_VEL
LIN {X 0,Y 573.631,Z 426.863,A -85,B 0,C 180,E1 -2090.624,E2 -2090.624} C_VEL
LIN {X 0,Y 573.528,Z 438.636,A -85,B 0,C 180,E1 -2091.267,E2 -2091.267} C_VEL
LIN {X 0,Y 573.405,Z 449.877,A -85,B 0,C 180,E1 -2092.046,E2 -2092.046} C_VEL
LIN {X 0,Y 573.267,Z 459.878,A -85,B 0,C 180,E1 -2092.907,E2 -2092.907} C_VEL
LIN {X 0,Y 573.137,Z 468.9,A -85,B 0,C 180,E1 -2093.869,E2 -2093.869} C_VEL
LIN {X 0,Y 573.098,Z 476.353,A -85,B 0,C 180,E1 -2094.841,E2 -2094.841} C_VEL
LIN {X 0,Y 573.067,Z 483.552,A -85,B 0,C 180,E1 -2096.004,E2 -2096.004} C_VEL
LIN {X 0,Y 573.008,Z 488.375,A -85,B 0,C 180,E1 -2096.988,E2 -2096.988} C_VEL
LIN {X 0,Y 572.969,Z 492.206,A -85,B 0,C 180,E1 -2097.975,E2 -2097.975} C_VEL
LIN {X 0,Y 572.992,Z 495.173,A -85,B 0,C 180,E1 -2098.978,E2 -2098.978} C_VEL
LIN {X 0,Y 572.946,Z 497.606,A -85,B 0,C 180,E1 -2100.193,E2 -2100.193} C_VEL
LIN {X 0,Y 572.959,Z 498.561,A -85,B 0,C 180,E1 -2101.009,E2 -2101.009} C_VEL
LIN {X 0,Y 572.952,Z 498.976,A -85,B 0,C 180,E1 -2102.18,E2 -2102.18} C_VEL
LIN {X 0,Y 572.965,Z 498.128,A -85,B 0,C 180,E1 -2103.502,E2 -2103.502} C_VEL
LIN {X 0,Y 572.965,Z 496.076,A -85,B 0,C 180,E1 -2104.732,E2 -2104.732} C_VEL
LIN {X 0,Y 573.001,Z 492.375,A -85,B 0,C 180,E1 -2106.066,E2 -2106.066} C_VEL
LIN {X 0,Y 573.017,Z 488.229,A -85,B 0,C 180,E1 -2107.134,E2 -2107.134} C_VEL
LIN {X 0,Y 573.075,Z 482.39,A -85,B 0,C 180,E1 -2108.29,E2 -2108.29} C_VEL
LIN {X 0,Y 573.113,Z 475.194,A -85,B 0,C 180,E1 -2109.415,E2 -2109.415} C_VEL
LIN {X 0,Y 573.199,Z 466.207,A -85,B 0,C 180,E1 -2110.528,E2 -2110.528} C_VEL
LIN {X 0,Y 573.299,Z 456.975,A -85,B 0,C 180,E1 -2111.45,E2 -2111.45} C_VEL
LIN {X 0,Y 573.37,Z 446.769,A -85,B 0,C 180,E1 -2112.281,E2 -2112.281} C_VEL
LIN {X 0,Y 573.461,Z 436.31,A -85,B 0,C 180,E1 -2112.965,E2 -2112.965} C_VEL
LIN {X 0,Y 573.609,Z 424.42,A -85,B 0,C 180,E1 -2113.578,E2 -2113.578} C_VEL
LIN {X 0,Y 573.768,Z 411.571,A -85,B 0,C 180,E1 -2114.074,E2 -2114.074} C_VEL
LIN {X 0,Y 573.716,Z 400.458,A -85,B 0,C 180,E1 -2114.38,E2 -2114.38} C_VEL
LIN {X 0,Y 572.902,Z 395.686,A -85,B 0,C 180,E1 -2114.498,E2 -2114.498} C_VEL
LIN {X 0,Y 572.952,Z 391.604,A -85,B 0,C 180,E1 -2117.573,E2 -2117.573} C_VEL
LIN {X 0,Y 572.915,Z 387.639,A -85,B 0,C 180,E1 -2120.607,E2 -2120.607} C_VEL
LIN {X 0,Y 572.956,Z 384.488,A -85,B 0,C 180,E1 -2123.055,E2 -2123.055} C_VEL
LIN {X 0,Y 572.955,Z 381.226,A -85,B 0,C 180,E1 -2125.65,E2 -2125.65} C_VEL
LIN {X 0,Y 573.03,Z 378.444,A -85,B 0,C 180,E1 -2128.171,E2 -2128.171} C_VEL
LIN {X 0,Y 573.064,Z 375.752,A -85,B 0,C 180,E1 -2130.623,E2 -2130.623} C_VEL
LIN {X 0,Y 573.099,Z 372.411,A -85,B 0,C 180,E1 -2133.533,E2 -2133.533} C_VEL
LIN {X 0,Y 573.101,Z 369.363,A -85,B 0,C 180,E1 -2136.129,E2 -2136.129} C_VEL
LIN {X 0,Y 573.224,Z 369.084,A -85,B 0,C 180,E1 -2137.662,E2 -2137.662} C_VEL
LIN {X 0,Y 573.251,Z 369.081,A -85,B 0,C 180,E1 -2139.923,E2 -2139.923} C_VEL
LIN {X 0,Y 573.255,Z 369.079,A -85,B 0,C 180,E1 -2142.989,E2 -2142.989} C_VEL
LIN {X 0,Y 573.267,Z 369.081,A -85,B 0,C 180,E1 -2145.807,E2 -2145.807} C_VEL
LIN {X 0,Y 573.277,Z 369.076,A -85,B 0,C 180,E1 -2148.734,E2 -2148.734} C_VEL
LIN {X 0,Y 573.285,Z 369.076,A -85,B 0,C 180,E1 -2151.54,E2 -2151.54} C_VEL
LIN {X 0,Y 573.286,Z 369.077,A -85,B 0,C 180,E1 -2154.372,E2 -2154.372} C_VEL
LIN {X 0,Y 573.306,Z 369.076,A -85,B 0,C 180,E1 -2157.892,E2 -2157.892} C_VEL
LIN {X 0,Y 573.332,Z 369.07,A -85,B 0,C 180,E1 -2160.702,E2 -2160.702} C_VEL
LIN {X 0,Y 573.233,Z 369.082,A -85,B 0,C 180,E1 -2163.514,E2 -2163.514} C_VEL
LIN {X 0,Y 573.285,Z 369.075,A -85,B 0,C 180,E1 -2165.628,E2 -2165.628} C_VEL
LIN {X 0,Y 573.282,Z 369.076,A -85,B 0,C 180,E1 -2168.46,E2 -2168.46} C_VEL
LIN {X 0,Y 573.293,Z 369.077,A -85,B 0,C 180,E1 -2171.312,E2 -2171.312} C_VEL
LIN {X 0,Y 573.274,Z 369.076,A -85,B 0,C 180,E1 -2174.425,E2 -2174.425} C_VEL
LIN {X 0,Y 573.254,Z 369.08,A -85,B 0,C 180,E1 -2177.112,E2 -2177.112} C_VEL
LIN {X 0,Y 573.247,Z 369.08,A -85,B 0,C 180,E1 -2180.077,E2 -2180.077} C_VEL
LIN {X 0,Y 573.228,Z 369.083,A -85,B 0,C 180,E1 -2183.1,E2 -2183.1} C_VEL
LIN {X 0,Y 573.252,Z 369.08,A -85,B 0,C 180,E1 -2185.41,E2 -2185.41} C_VEL
LIN {X 0,Y 573.259,Z 369.08,A -85,B 0,C 180,E1 -2188.032,E2 -2188.032} C_VEL
LIN {X 0,Y 573.222,Z 369.084,A -85,B 0,C 180,E1 -2190.883,E2 -2190.883} C_VEL
LIN {X 0,Y 573.235,Z 369.082,A -85,B 0,C 180,E1 -2193.521,E2 -2193.521} C_VEL
LIN {X 0,Y 573.211,Z 369.085,A -85,B 0,C 180,E1 -2196.052,E2 -2196.052} C_VEL
LIN {X 0,Y 573.246,Z 369.081,A -85,B 0,C 180,E1 -2198.701,E2 -2198.701} C_VEL
LIN {X 0,Y 573.25,Z 369.082,A -85,B 0,C 180,E1 -2201.596,E2 -2201.596} C_VEL
LIN {X 0,Y 573.233,Z 369.082,A -85,B 0,C 180,E1 -2204.334,E2 -2204.334} C_VEL
LIN {X 0,Y 573.238,Z 369.083,A -85,B 0,C 180,E1 -2207.359,E2 -2207.359} C_VEL
LIN {X 0,Y 573.245,Z 369.081,A -85,B 0,C 180,E1 -2210.394,E2 -2210.394} C_VEL
LIN {X 0,Y 573.281,Z 369.122,A -85,B 0,C 180,E1 -2213.245,E2 -2213.245} C_VEL
LIN {X 0,Y 573.781,Z 372.595,A -85,B 0,C 180,E1 -2214.423,E2 -2214.423} C_VEL
LIN {X 0,Y 573.705,Z 380.538,A -85,B 0,C 180,E1 -2216.967,E2 -2216.967} C_VEL
LIN {X 0,Y 573.585,Z 388.524,A -85,B 0,C 180,E1 -2219.45,E2 -2219.45} C_VEL
LIN {X 0,Y 573.482,Z 397.748,A -85,B 0,C 180,E1 -2222.246,E2 -2222.246} C_VEL
LIN {X 0,Y 573.426,Z 407.363,A -85,B 0,C 180,E1 -2225.088,E2 -2225.088} C_VEL
LIN {X 0,Y 573.351,Z 417.606,A -85,B 0,C 180,E1 -2228.046,E2 -2228.046} C_VEL
LIN {X 0,Y 573.227,Z 428.33,A -85,B 0,C 180,E1 -2231.078,E2 -2231.078} C_VEL
LIN {X 0,Y 573.165,Z 438.788,A -85,B 0,C 180,E1 -2233.985,E2 -2233.985} C_VEL
LIN {X 0,Y 573.098,Z 449.379,A -85,B 0,C 180,E1 -2236.887,E2 -2236.887} C_VEL
LIN {X 0,Y 573.085,Z 451.53,A -85,B 0,C 180,E1 -2237.472,E2 -2237.472} C_VEL
LIN {X 0,Y 573.876,Z 457.234,A -85,B 0,C 180,E1 -2237.602,E2 -2237.602} C_VEL
LIN {X 0,Y 573.781,Z 470.499,A -85,B 0,C 180,E1 -2237.937,E2 -2237.937} C_VEL
LIN {X 0,Y 573.629,Z 482.802,A -85,B 0,C 180,E1 -2238.395,E2 -2238.395} C_VEL
LIN {X 0,Y 573.516,Z 494.441,A -85,B 0,C 180,E1 -2238.974,E2 -2238.974} C_VEL
LIN {X 0,Y 573.452,Z 505.478,A -85,B 0,C 180,E1 -2239.675,E2 -2239.675} C_VEL
LIN {X 0,Y 573.308,Z 515.647,A -85,B 0,C 180,E1 -2240.474,E2 -2240.474} C_VEL
LIN {X 0,Y 573.215,Z 524.787,A -85,B 0,C 180,E1 -2241.362,E2 -2241.362} C_VEL
LIN {X 0,Y 573.142,Z 533.69,A -85,B 0,C 180,E1 -2242.425,E2 -2242.425} C_VEL
LIN {X 0,Y 573.051,Z 540.405,A -85,B 0,C 180,E1 -2243.415,E2 -2243.415} C_VEL
LIN {X 0,Y 573.07,Z 545.68,A -85,B 0,C 180,E1 -2244.37,E2 -2244.37} C_VEL
LIN {X 0,Y 573.028,Z 550.371,A -85,B 0,C 180,E1 -2245.427,E2 -2245.427} C_VEL
LIN {X 0,Y 573.022,Z 553.956,A -85,B 0,C 180,E1 -2246.484,E2 -2246.484} C_VEL
LIN {X 0,Y 572.959,Z 555.808,A -85,B 0,C 180,E1 -2247.188,E2 -2247.188} C_VEL
LIN {X 0,Y 572.94,Z 557.2,A -85,B 0,C 180,E1 -2247.891,E2 -2247.891} C_VEL
LIN {X 0,Y 572.94,Z 558.784,A -85,B 0,C 180,E1 -2249.297,E2 -2249.297} C_VEL
LIN {X 0,Y 572.938,Z 559,A -85,B 0,C 180,E1 -2250,E2 -2250} C_VEL
LIN {X 0,Y 572.946,Z 558.185,A -85,B 0,C 180,E1 -2251.406,E2 -2251.406} C_VEL
LIN {X 0,Y 572.939,Z 557.202,A -85,B 0,C 180,E1 -2252.109,E2 -2252.109} C_VEL
LIN {X 0,Y 572.959,Z 555.81,A -85,B 0,C 180,E1 -2252.812,E2 -2252.812} C_VEL
LIN {X 0,Y 573.015,Z 552.897,A -85,B 0,C 180,E1 -2253.868,E2 -2253.868} C_VEL
LIN {X 0,Y 572.963,Z 548.951,A -85,B 0,C 180,E1 -2254.925,E2 -2254.925} C_VEL
LIN {X 0,Y 573.064,Z 542.879,A -85,B 0,C 180,E1 -2256.16,E2 -2256.16} C_VEL
LIN {X 0,Y 573.119,Z 536.239,A -85,B 0,C 180,E1 -2257.22,E2 -2257.22} C_VEL
LIN {X 0,Y 573.2,Z 527.993,A -85,B 0,C 180,E1 -2258.283,E2 -2258.283} C_VEL
LIN {X 0,Y 573.287,Z 519.541,A -85,B 0,C 180,E1 -2259.17,E2 -2259.17} C_VEL
LIN {X 0,Y 573.417,Z 509.099,A -85,B 0,C 180,E1 -2260.058,E2 -2260.058} C_VEL
LIN {X 0,Y 573.522,Z 497.536,A -85,B 0,C 180,E1 -2260.847,E2 -2260.847} C_VEL
LIN {X 0,Y 573.61,Z 485.888,A -85,B 0,C 180,E1 -2261.466,E2 -2261.466} C_VEL
LIN {X 0,Y 573.733,Z 473.188,A -85,B 0,C 180,E1 -2261.974,E2 -2261.974} C_VEL
LIN {X 0,Y 573.868,Z 460.539,A -85,B 0,C 180,E1 -2262.33,E2 -2262.33} C_VEL
LIN {X 0,Y 573.574,Z 454.673,A -85,B 0,C 180,E1 -2262.455,E2 -2262.455} C_VEL
LIN {X 0,Y 573.085,Z 451.532,A -85,B 0,C 180,E1 -2262.527,E2 -2262.527} C_VEL
LIN {X 0,Y 573.157,Z 441.437,A -85,B 0,C 180,E1 -2265.285,E2 -2265.285} C_VEL
LIN {X 0,Y 573.216,Z 430.846,A -85,B 0,C 180,E1 -2268.218,E2 -2268.218} C_VEL
LIN {X 0,Y 573.299,Z 421.579,A -85,B 0,C 180,E1 -2270.824,E2 -2270.824} C_VEL
LIN {X 0,Y 573.353,Z 412.313,A -85,B 0,C 180,E1 -2273.476,E2 -2273.476} C_VEL
LIN {X 0,Y 573.454,Z 403.045,A -85,B 0,C 180,E1 -2276.18,E2 -2276.18} C_VEL
LIN {X 0,Y 573.498,Z 393.778,A -85,B 0,C 180,E1 -2278.95,E2 -2278.95} C_VEL
LIN {X 0,Y 573.631,Z 385.835,A -85,B 0,C 180,E1 -2281.378,E2 -2281.378} C_VEL
LIN {X 0,Y 573.776,Z 376.568,A -85,B 0,C 180,E1 -2284.293,E2 -2284.293} C_VEL
LIN {X 0,Y 573.647,Z 371.205,A -85,B 0,C 180,E1 -2286.041,E2 -2286.041} C_VEL
LIN {X 0,Y 573.265,Z 369.078,A -85,B 0,C 180,E1 -2286.811,E2 -2286.811} C_VEL
LIN {X 0,Y 573.236,Z 369.085,A -85,B 0,C 180,E1 -2289.607,E2 -2289.607} C_VEL
LIN {X 0,Y 573.239,Z 369.083,A -85,B 0,C 180,E1 -2292.641,E2 -2292.641} C_VEL
LIN {X 0,Y 573.23,Z 369.083,A -85,B 0,C 180,E1 -2295.666,E2 -2295.666} C_VEL
LIN {X 0,Y 573.239,Z 369.084,A -85,B 0,C 180,E1 -2298.544,E2 -2298.544} C_VEL
LIN {X 0,Y 573.243,Z 369.081,A -85,B 0,C 180,E1 -2301.298,E2 -2301.298} C_VEL
LIN {X 0,Y 573.259,Z 369.081,A -85,B 0,C 180,E1 -2304.01,E2 -2304.01} C_VEL
LIN {X 0,Y 573.278,Z 369.077,A -85,B 0,C 180,E1 -2306.518,E2 -2306.518} C_VEL
LIN {X 0,Y 573.231,Z 369.083,A -85,B 0,C 180,E1 -2309.115,E2 -2309.115} C_VEL
LIN {X 0,Y 573.258,Z 369.08,A -85,B 0,C 180,E1 -2311.967,E2 -2311.967} C_VEL
LIN {X 0,Y 573.247,Z 369.08,A -85,B 0,C 180,E1 -2314.59,E2 -2314.59} C_VEL
LIN {X 0,Y 573.23,Z 369.082,A -85,B 0,C 180,E1 -2317.662,E2 -2317.662} C_VEL
LIN {X 0,Y 573.25,Z 369.08,A -85,B 0,C 180,E1 -2319.923,E2 -2319.923} C_VEL
LIN {X 0,Y 573.256,Z 369.08,A -85,B 0,C 180,E1 -2322.988,E2 -2322.988} C_VEL
LIN {X 0,Y 573.264,Z 369.078,A -85,B 0,C 180,E1 -2325.807,E2 -2325.807} C_VEL
LIN {X 0,Y 573.274,Z 369.077,A -85,B 0,C 180,E1 -2328.734,E2 -2328.734} C_VEL
LIN {X 0,Y 573.298,Z 369.076,A -85,B 0,C 180,E1 -2331.541,E2 -2331.541} C_VEL
LIN {X 0,Y 573.282,Z 369.076,A -85,B 0,C 180,E1 -2334.372,E2 -2334.372} C_VEL
LIN {X 0,Y 573.301,Z 369.073,A -85,B 0,C 180,E1 -2337.892,E2 -2337.892} C_VEL
LIN {X 0,Y 573.333,Z 369.071,A -85,B 0,C 180,E1 -2340.702,E2 -2340.702} C_VEL
LIN {X 0,Y 573.234,Z 369.082,A -85,B 0,C 180,E1 -2343.515,E2 -2343.515} C_VEL
LIN {X 0,Y 573.285,Z 369.075,A -85,B 0,C 180,E1 -2345.628,E2 -2345.628} C_VEL
LIN {X 0,Y 573.299,Z 369.075,A -85,B 0,C 180,E1 -2348.459,E2 -2348.459} C_VEL
LIN {X 0,Y 573.29,Z 369.076,A -85,B 0,C 180,E1 -2351.312,E2 -2351.312} C_VEL
LIN {X 0,Y 573.272,Z 369.077,A -85,B 0,C 180,E1 -2354.425,E2 -2354.425} C_VEL
LIN {X 0,Y 573.251,Z 369.082,A -85,B 0,C 180,E1 -2357.112,E2 -2357.112} C_VEL
LIN {X 0,Y 573.25,Z 369.08,A -85,B 0,C 180,E1 -2360.077,E2 -2360.077} C_VEL
